KUKA KRL program: EPS_2_251692_SAMH01_A_20251205090654.src

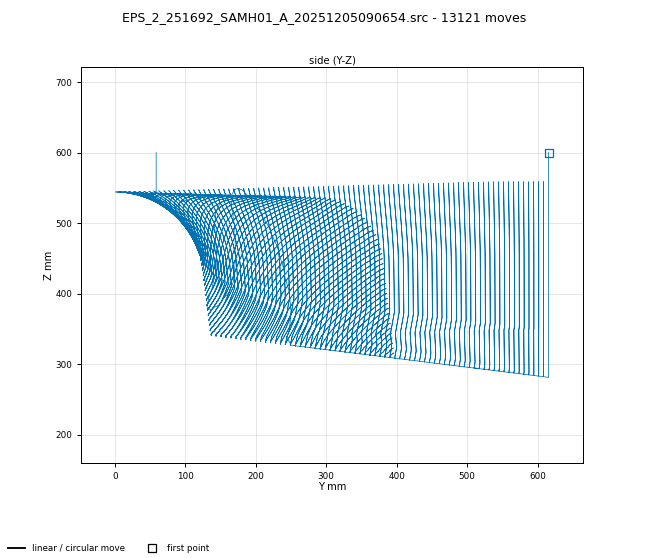
[picture p0: tool path of EPS_2_251692_SAMH01_A_20251205090654.src, 13121 of 13123 moves have a stored position in this frame; points joined in program order, loops and branches not executed]
&ACCESS RVP
&REL 4
&COMMENT QRS 19112012
&PARAM EDITMASK = *
DEF PART()
EXT BAS (BAS_COMMAND :IN,REAL :IN )
INT I
BAS (#INITMOV,0 )

;KUKA QRS Post kuka4.cps  Date:22-06-2017 !

File_ID=2943

QRS_PRE_INIT()

;Init var - Until changes are made in qrs_pre_init
Outlet_Square_prg=0
Inlet_1_Square_prg=0
Inlet_2_Square_prg=0
Inlet_3_Square_prg=0
Inlet_4_Square_prg=0
Inlet_5_Square_prg=0

Outlet_1={X 0.000, Y 535.490, Z 458.500, B 0.000, E1 0.000 }
Inlet_1={X 0.000, Y 556.400, Z 433.500, B 0.000, E1 180.000 }
Outlet_1_type=201
Inlet_1_type=0
;QRS#1=Sidecore dimensions
;QRS#2=200-8" PVC SDR 35
;QRS#3=DeadEnd 201
;QRS#4=
;QRS#5=
;QRS#6=
;QRS#7=
;QRS#8=
;QRS#9=12-08 PSX
;QRS#10=

;QRS#11=
;QRS#12=
;QRS#13=
;QRS#14=
;QRS#15=
;QRS#16=1220x127x838 2,75'
;QRS#17=EPS Height
;QRS#18=559
;QRS#19=*
;QRS#20= UPDATED VERSION 22-06-2017
;QRS#21=*
Outlet_Square=0100
Inlet_1_Square=00
Inlet_2_Square=0
Inlet_3_Square=0
Inlet_4_Square=0
Inlet_5_Square=0
Mill_Square=1
Outlet_Square_Prg=204
Inlet_1_Square_prg=0

QRS_INIT()

$ADVANCE=5

; T1
PTP {E1 173.595,E2 173.595}
PTP {X 0,Y 615.506,A -85,B 0,C 180,E1 173.595,E2 173.595,E3 0,E4 0,E5 0,E6 0}
QRS_SPEED_INIT()
LIN {X 0,Y 615.506,Z 600,A -85,B 0,C 180,E1 173.595,E2 173.595,E3 0,E4 0,E5 0,E6 0} C_VEL
LIN {X 0,Y 615.506,Z 291.363,A -85,B 0,C 180,E1 173.595,E2 173.595} C_VEL
LIN {X 0,Y 615.506,Z 283.186,A -85,B 0,C 180,E1 173.595,E2 173.595} C_VEL
LIN {X 0,Y 615.49,Z 281.186,A -85,B 0,C 180,E1 173.408,E2 173.408} C_VEL
LIN {X 0,Y 615.486,Z 281.199,A -85,B 0,C 180,E1 170.802,E2 170.802} C_VEL
LIN {X 0,Y 615.467,Z 281.188,A -85,B 0,C 180,E1 168.139,E2 168.139} C_VEL
LIN {X 0,Y 615.487,Z 281.188,A -85,B 0,C 180,E1 165.451,E2 165.451} C_VEL
LIN {X 0,Y 615.474,Z 281.196,A -85,B 0,C 180,E1 162.73,E2 162.73} C_VEL
LIN {X 0,Y 615.487,Z 281.182,A -85,B 0,C 180,E1 159.968,E2 159.968} C_VEL
LIN {X 0,Y 615.487,Z 281.2,A -85,B 0,C 180,E1 157.156,E2 157.156} C_VEL
LIN {X 0,Y 615.469,Z 281.189,A -85,B 0,C 180,E1 154.432,E2 154.432} C_VEL
LIN {X 0,Y 615.482,Z 281.184,A -85,B 0,C 180,E1 152.085,E2 152.085} C_VEL
LIN {X 0,Y 615.489,Z 281.198,A -85,B 0,C 180,E1 149.081,E2 149.081} C_VEL
LIN {X 0,Y 615.472,Z 281.187,A -85,B 0,C 180,E1 146.466,E2 146.466} C_VEL
LIN {X 0,Y 615.492,Z 281.181,A -85,B 0,C 180,E1 144.164,E2 144.164} C_VEL
LIN {X 0,Y 615.485,Z 281.186,A -85,B 0,C 180,E1 141.932,E2 141.932} C_VEL
LIN {X 0,Y 615.485,Z 281.201,A -85,B 0,C 180,E1 139.394,E2 139.394} C_VEL
LIN {X 0,Y 615.471,Z 281.189,A -85,B 0,C 180,E1 136.754,E2 136.754} C_VEL
LIN {X 0,Y 615.486,Z 281.186,A -85,B 0,C 180,E1 133.998,E2 133.998} C_VEL
LIN {X 0,Y 615.497,Z 281.199,A -85,B 0,C 180,E1 131.472,E2 131.472} C_VEL
LIN {X 0,Y 615.472,Z 281.19,A -85,B 0,C 180,E1 128.904,E2 128.904} C_VEL
LIN {X 0,Y 615.484,Z 281.183,A -85,B 0,C 180,E1 126.424,E2 126.424} C_VEL
LIN {X 0,Y 615.495,Z 281.201,A -85,B 0,C 180,E1 123.536,E2 123.536} C_VEL
LIN {X 0,Y 615.474,Z 281.188,A -85,B 0,C 180,E1 120.92,E2 120.92} C_VEL
LIN {X 0,Y 615.491,Z 281.182,A -85,B 0,C 180,E1 118.452,E2 118.452} C_VEL
LIN {X 0,Y 615.492,Z 281.199,A -85,B 0,C 180,E1 115.571,E2 115.571} C_VEL
LIN {X 0,Y 615.48,Z 281.184,A -85,B 0,C 180,E1 112.844,E2 112.844} C_VEL
LIN {X 0,Y 615.483,Z 281.193,A -85,B 0,C 180,E1 110.032,E2 110.032} C_VEL
LIN {X 0,Y 615.475,Z 281.19,A -85,B 0,C 180,E1 107.27,E2 107.27} C_VEL
LIN {X 0,Y 615.482,Z 281.185,A -85,B 0,C 180,E1 104.549,E2 104.549} C_VEL
LIN {X 0,Y 615.486,Z 281.202,A -85,B 0,C 180,E1 101.861,E2 101.861} C_VEL
LIN {X 0,Y 615.479,Z 281.187,A -85,B 0,C 180,E1 99.199,E2 99.199} C_VEL
LIN {X 0,Y 615.479,Z 281.187,A -85,B 0,C 180,E1 96.557,E2 96.557} C_VEL
LIN {X 0,Y 615.486,Z 281.203,A -85,B 0,C 180,E1 93.928,E2 93.928} C_VEL
LIN {X 0,Y 615.48,Z 281.186,A -85,B 0,C 180,E1 91.309,E2 91.309} C_VEL
LIN {X 0,Y 615.48,Z 281.186,A -85,B 0,C 180,E1 88.691,E2 88.691} C_VEL
LIN {X 0,Y 615.486,Z 281.203,A -85,B 0,C 180,E1 86.072,E2 86.072} C_VEL
LIN {X 0,Y 615.48,Z 281.186,A -85,B 0,C 180,E1 83.424,E2 83.424} C_VEL
LIN {X 0,Y 615.479,Z 281.187,A -85,B 0,C 180,E1 80.801,E2 80.801} C_VEL
LIN {X 0,Y 615.486,Z 281.202,A -85,B 0,C 180,E1 78.139,E2 78.139} C_VEL
LIN {X 0,Y 615.482,Z 281.185,A -85,B 0,C 180,E1 75.451,E2 75.451} C_VEL
LIN {X 0,Y 615.475,Z 281.19,A -85,B 0,C 180,E1 72.73,E2 72.73} C_VEL
LIN {X 0,Y 615.483,Z 281.193,A -85,B 0,C 180,E1 69.968,E2 69.968} C_VEL
LIN {X 0,Y 615.481,Z 281.184,A -85,B 0,C 180,E1 67.156,E2 67.156} C_VEL
LIN {X 0,Y 615.495,Z 281.199,A -85,B 0,C 180,E1 64.285,E2 64.285} C_VEL
LIN {X 0,Y 615.483,Z 281.183,A -85,B 0,C 180,E1 61.342,E2 61.342} C_VEL
LIN {X 0,Y 615.473,Z 281.191,A -85,B 0,C 180,E1 58.915,E2 58.915} C_VEL
LIN {X 0,Y 615.495,Z 281.201,A -85,B 0,C 180,E1 56.464,E2 56.464} C_VEL
LIN {X 0,Y 615.484,Z 281.183,A -85,B 0,C 180,E1 53.576,E2 53.576} C_VEL
LIN {X 0,Y 615.474,Z 281.193,A -85,B 0,C 180,E1 50.939,E2 50.939} C_VEL
LIN {X 0,Y 615.497,Z 281.199,A -85,B 0,C 180,E1 48.528,E2 48.528} C_VEL
LIN {X 0,Y 615.492,Z 281.183,A -85,B 0,C 180,E1 45.852,E2 45.852} C_VEL
LIN {X 0,Y 615.473,Z 281.193,A -85,B 0,C 180,E1 43.047,E2 43.047} C_VEL
LIN {X 0,Y 615.485,Z 281.201,A -85,B 0,C 180,E1 40.606,E2 40.606} C_VEL
LIN {X 0,Y 615.485,Z 281.185,A -85,B 0,C 180,E1 38.013,E2 38.013} C_VEL
LIN {X 0,Y 615.476,Z 281.185,A -85,B 0,C 180,E1 35.616,E2 35.616} C_VEL
LIN {X 0,Y 615.47,Z 281.192,A -85,B 0,C 180,E1 33.237,E2 33.237} C_VEL
LIN {X 0,Y 615.489,Z 281.198,A -85,B 0,C 180,E1 30.919,E2 30.919} C_VEL
LIN {X 0,Y 615.484,Z 281.183,A -85,B 0,C 180,E1 27.915,E2 27.915} C_VEL
LIN {X 0,Y 615.467,Z 281.189,A -85,B 0,C 180,E1 25.568,E2 25.568} C_VEL
LIN {X 0,Y 615.487,Z 281.2,A -85,B 0,C 180,E1 22.844,E2 22.844} C_VEL
LIN {X 0,Y 615.487,Z 281.182,A -85,B 0,C 180,E1 20.032,E2 20.032} C_VEL
LIN {X 0,Y 615.474,Z 281.196,A -85,B 0,C 180,E1 17.27,E2 17.27} C_VEL
LIN {X 0,Y 615.487,Z 281.188,A -85,B 0,C 180,E1 14.549,E2 14.549} C_VEL
LIN {X 0,Y 615.467,Z 281.188,A -85,B 0,C 180,E1 11.861,E2 11.861} C_VEL
LIN {X 0,Y 615.486,Z 281.199,A -85,B 0,C 180,E1 9.198,E2 9.198} C_VEL
LIN {X 0,Y 615.491,Z 281.185,A -85,B 0,C 180,E1 6.556,E2 6.556} C_VEL
LIN {X 0,Y 615.464,Z 281.189,A -85,B 0,C 180,E1 3.928,E2 3.928} C_VEL
LIN {X 0,Y 615.485,Z 281.2,A -85,B 0,C 180,E1 1.308,E2 1.308} C_VEL
LIN {X 0,Y 615.491,Z 281.186,A -85,B 0,C 180,E1 -1.309,E2 -1.309} C_VEL
LIN {X 0,Y 615.465,Z 281.188,A -85,B 0,C 180,E1 -3.929,E2 -3.929} C_VEL
LIN {X 0,Y 615.483,Z 281.2,A -85,B 0,C 180,E1 -6.586,E2 -6.586} C_VEL
LIN {X 0,Y 615.492,Z 281.185,A -85,B 0,C 180,E1 -9.199,E2 -9.199} C_VEL
LIN {X 0,Y 615.462,Z 281.19,A -85,B 0,C 180,E1 -11.862,E2 -11.862} C_VEL
LIN {X 0,Y 615.487,Z 281.202,A -85,B 0,C 180,E1 -14.549,E2 -14.549} C_VEL
LIN {X 0,Y 615.491,Z 281.183,A -85,B 0,C 180,E1 -17.271,E2 -17.271} C_VEL
LIN {X 0,Y 615.463,Z 281.194,A -85,B 0,C 180,E1 -20.034,E2 -20.034} C_VEL
LIN {X 0,Y 615.491,Z 281.19,A -85,B 0,C 180,E1 -22.845,E2 -22.845} C_VEL
LIN {X 0,Y 615.458,Z 281.189,A -85,B 0,C 180,E1 -25.566,E2 -25.566} C_VEL
LIN {X 0,Y 615.462,Z 281.194,A -85,B 0,C 180,E1 -27.917,E2 -27.917} C_VEL
LIN {X 0,Y 615.474,Z 281.199,A -85,B 0,C 180,E1 -30.161,E2 -30.161} C_VEL
LIN {X 0,Y 615.494,Z 281.197,A -85,B 0,C 180,E1 -32.457,E2 -32.457} C_VEL
LIN {X 0,Y 615.494,Z 281.186,A -85,B 0,C 180,E1 -34.815,E2 -34.815} C_VEL
LIN {X 0,Y 615.466,Z 281.187,A -85,B 0,C 180,E1 -37.244,E2 -37.244} C_VEL
LIN {X 0,Y 615.485,Z 281.198,A -85,B 0,C 180,E1 -40.09,E2 -40.09} C_VEL
LIN {X 0,Y 615.472,Z 281.186,A -85,B 0,C 180,E1 -43.047,E2 -43.047} C_VEL
LIN {X 0,Y 615.469,Z 281.197,A -85,B 0,C 180,E1 -45.85,E2 -45.85} C_VEL
LIN {X 0,Y 615.493,Z 281.188,A -85,B 0,C 180,E1 -48.528,E2 -48.528} C_VEL
LIN {X 0,Y 615.46,Z 281.188,A -85,B 0,C 180,E1 -51.095,E2 -51.095} C_VEL
LIN {X 0,Y 615.459,Z 281.195,A -85,B 0,C 180,E1 -53.574,E2 -53.574} C_VEL
LIN {X 0,Y 615.496,Z 281.187,A -85,B 0,C 180,E1 -56.465,E2 -56.465} C_VEL
LIN {X 0,Y 615.455,Z 281.19,A -85,B 0,C 180,E1 -59.079,E2 -59.079} C_VEL
LIN {X 0,Y 615.463,Z 281.196,A -85,B 0,C 180,E1 -61.554,E2 -61.554} C_VEL
LIN {X 0,Y 615.498,Z 281.185,A -85,B 0,C 180,E1 -64.43,E2 -64.43} C_VEL
LIN {X 0,Y 615.497,Z 281.361,A -85,B 0,C 180,E1 -65.958,E2 -65.958} C_VEL
LIN {X 0,Y 615.494,Z 296.441,A -85,B 0,C 180,E1 -68.569,E2 -68.569} C_VEL
LIN {X 0,Y 615.488,Z 313.211,A -85,B 0,C 180,E1 -71.396,E2 -71.396} C_VEL
LIN {X 0,Y 615.498,Z 330.499,A -85,B 0,C 180,E1 -74.265,E2 -74.265} C_VEL
LIN {X 0,Y 615.496,Z 347.73,A -85,B 0,C 180,E1 -77.072,E2 -77.072} C_VEL
LIN {X 0,Y 615.493,Z 349.262,A -85,B 0,C 180,E1 -77.156,E2 -77.156} C_VEL
LIN {X 0,Y 615.497,Z 454.843,A -85,B 0,C 180,E1 -78.411,E2 -78.411} C_VEL
LIN {X 0,Y 615.499,Z 467.352,A -85,B 0,C 180,E1 -78.682,E2 -78.682} C_VEL
LIN {X 0,Y 615.496,Z 480.501,A -85,B 0,C 180,E1 -79.109,E2 -79.109} C_VEL
LIN {X 0,Y 615.486,Z 492.482,A -85,B 0,C 180,E1 -79.64,E2 -79.64} C_VEL
LIN {X 0,Y 615.493,Z 503.998,A -85,B 0,C 180,E1 -80.304,E2 -80.304} C_VEL
LIN {X 0,Y 615.499,Z 514.344,A -85,B 0,C 180,E1 -81.05,E2 -81.05} C_VEL
LIN {X 0,Y 615.497,Z 522.814,A -85,B 0,C 180,E1 -81.794,E2 -81.794} C_VEL
LIN {X 0,Y 615.498,Z 530.608,A -85,B 0,C 180,E1 -82.62,E2 -82.62} C_VEL
LIN {X 0,Y 615.496,Z 538.204,A -85,B 0,C 180,E1 -83.608,E2 -83.608} C_VEL
LIN {X 0,Y 615.498,Z 545.205,A -85,B 0,C 180,E1 -84.759,E2 -84.759} C_VEL
LIN {X 0,Y 615.493,Z 549.852,A -85,B 0,C 180,E1 -85.744,E2 -85.744} C_VEL
LIN {X 0,Y 615.495,Z 553.399,A -85,B 0,C 180,E1 -86.727,E2 -86.727} C_VEL
LIN {X 0,Y 615.497,Z 555.233,A -85,B 0,C 180,E1 -87.382,E2 -87.382} C_VEL
LIN {X 0,Y 615.499,Z 556.608,A -85,B 0,C 180,E1 -88.037,E2 -88.037} C_VEL
LIN {X 0,Y 615.496,Z 558.174,A -85,B 0,C 180,E1 -89.346,E2 -89.346} C_VEL
LIN {X 0,Y 615.494,Z 558.389,A -85,B 0,C 180,E1 -90,E2 -90} C_VEL
LIN {X 0,Y 615.496,Z 557.58,A -85,B 0,C 180,E1 -91.309,E2 -91.309} C_VEL
LIN {X 0,Y 615.499,Z 556.608,A -85,B 0,C 180,E1 -91.963,E2 -91.963} C_VEL
LIN {X 0,Y 615.497,Z 555.233,A -85,B 0,C 180,E1 -92.618,E2 -92.618} C_VEL
LIN {X 0,Y 615.496,Z 552.35,A -85,B 0,C 180,E1 -93.601,E2 -93.601} C_VEL
LIN {X 0,Y 615.498,Z 548.442,A -85,B 0,C 180,E1 -94.584,E2 -94.584} C_VEL
LIN {X 0,Y 615.499,Z 543.406,A -85,B 0,C 180,E1 -95.57,E2 -95.57} C_VEL
LIN {X 0,Y 615.497,Z 536.87,A -85,B 0,C 180,E1 -96.583,E2 -96.583} C_VEL
LIN {X 0,Y 615.497,Z 529.135,A -85,B 0,C 180,E1 -97.545,E2 -97.545} C_VEL
LIN {X 0,Y 615.498,Z 521.047,A -85,B 0,C 180,E1 -98.371,E2 -98.371} C_VEL
LIN {X 0,Y 615.499,Z 511.17,A -85,B 0,C 180,E1 -99.198,E2 -99.198} C_VEL
LIN {X 0,Y 615.493,Z 499.985,A -85,B 0,C 180,E1 -99.945,E2 -99.945} C_VEL
LIN {X 0,Y 615.489,Z 489.027,A -85,B 0,C 180,E1 -100.527,E2 -100.527} C_VEL
LIN {X 0,Y 615.499,Z 476.422,A -85,B 0,C 180,E1 -101.042,E2 -101.042} C_VEL
LIN {X 0,Y 615.499,Z 464.075,A -85,B 0,C 180,E1 -101.401,E2 -101.401} C_VEL
LIN {X 0,Y 615.498,Z 450.483,A -85,B 0,C 180,E1 -101.651,E2 -101.651} C_VEL
LIN {X 0,Y 615.494,Z 348.55,A -85,B 0,C 180,E1 -102.865,E2 -102.865} C_VEL
LIN {X 0,Y 615.495,Z 346.987,A -85,B 0,C 180,E1 -103.033,E2 -103.033} C_VEL
LIN {X 0,Y 615.495,Z 329.466,A -85,B 0,C 180,E1 -105.905,E2 -105.905} C_VEL
LIN {X 0,Y 615.487,Z 312.962,A -85,B 0,C 180,E1 -108.646,E2 -108.646} C_VEL
LIN {X 0,Y 615.494,Z 296.441,A -85,B 0,C 180,E1 -111.431,E2 -111.431} C_VEL
LIN {X 0,Y 615.497,Z 281.361,A -85,B 0,C 180,E1 -114.042,E2 -114.042} C_VEL
LIN {X 0,Y 615.465,Z 281.196,A -85,B 0,C 180,E1 -116.444,E2 -116.444} C_VEL
LIN {X 0,Y 615.453,Z 281.193,A -85,B 0,C 180,E1 -118.659,E2 -118.659} C_VEL
LIN {X 0,Y 615.462,Z 281.188,A -85,B 0,C 180,E1 -121.082,E2 -121.082} C_VEL
LIN {X 0,Y 615.491,Z 281.201,A -85,B 0,C 180,E1 -124.021,E2 -124.021} C_VEL
LIN {X 0,Y 615.459,Z 281.195,A -85,B 0,C 180,E1 -126.426,E2 -126.426} C_VEL
LIN {X 0,Y 615.47,Z 281.187,A -85,B 0,C 180,E1 -129.06,E2 -129.06} C_VEL
LIN {X 0,Y 615.478,Z 281.198,A -85,B 0,C 180,E1 -132.079,E2 -132.079} C_VEL
LIN {X 0,Y 615.47,Z 281.196,A -85,B 0,C 180,E1 -134.15,E2 -134.15} C_VEL
LIN {X 0,Y 615.472,Z 281.186,A -85,B 0,C 180,E1 -136.953,E2 -136.953} C_VEL
LIN {X 0,Y 615.485,Z 281.198,A -85,B 0,C 180,E1 -139.91,E2 -139.91} C_VEL
LIN {X 0,Y 615.466,Z 281.187,A -85,B 0,C 180,E1 -142.756,E2 -142.756} C_VEL
LIN {X 0,Y 615.492,Z 281.189,A -85,B 0,C 180,E1 -145.297,E2 -145.297} C_VEL
LIN {X 0,Y 615.494,Z 281.201,A -85,B 0,C 180,E1 -147.666,E2 -147.666} C_VEL
LIN {X 0,Y 615.459,Z 281.193,A -85,B 0,C 180,E1 -150.208,E2 -150.208} C_VEL
LIN {X 0,Y 615.497,Z 281.183,A -85,B 0,C 180,E1 -152.951,E2 -152.951} C_VEL
LIN {X 0,Y 615.482,Z 281.198,A -85,B 0,C 180,E1 -155.727,E2 -155.727} C_VEL
LIN {X 0,Y 615.469,Z 281.196,A -85,B 0,C 180,E1 -157.863,E2 -157.863} C_VEL
LIN {X 0,Y 615.483,Z 281.184,A -85,B 0,C 180,E1 -160.662,E2 -160.662} C_VEL
LIN {X 0,Y 615.482,Z 281.2,A -85,B 0,C 180,E1 -163.566,E2 -163.566} C_VEL
LIN {X 0,Y 615.461,Z 281.19,A -85,B 0,C 180,E1 -166.125,E2 -166.125} C_VEL
LIN {X 0,Y 615.493,Z 281.185,A -85,B 0,C 180,E1 -168.807,E2 -168.807} C_VEL
LIN {X 0,Y 615.487,Z 281.198,A -85,B 0,C 180,E1 -171.463,E2 -171.463} C_VEL
LIN {X 0,Y 615.464,Z 281.188,A -85,B 0,C 180,E1 -174.101,E2 -174.101} C_VEL
LIN {X 0,Y 615.489,Z 281.186,A -85,B 0,C 180,E1 -176.727,E2 -176.727} C_VEL
LIN {X 0,Y 615.489,Z 281.198,A -85,B 0,C 180,E1 -179.345,E2 -179.345} C_VEL
LIN {X 0,Y 615.465,Z 281.189,A -85,B 0,C 180,E1 -181.963,E2 -181.963} C_VEL
LIN {X 0,Y 615.492,Z 281.185,A -85,B 0,C 180,E1 -184.584,E2 -184.584} C_VEL
LIN {X 0,Y 615.49,Z 281.186,A -85,B 0,C 180,E1 -186.592,E2 -186.592} C_VEL
LIN {X 0,Y 614.813,Z 281.345,A -85,B 0,C 180,E1 -187.138,E2 -187.138} C_VEL
LIN {X 0,Y 611.978,Z 281.748,A -85,B 0,C 180,E1 -188.024,E2 -188.024} C_VEL
LIN {X 0,Y 609.584,Z 282.063,A -85,B 0,C 180,E1 -188.736,E2 -188.736} C_VEL
LIN {X 0,Y 608.544,Z 282.183,A -85,B 0,C 180,E1 -189.286,E2 -189.286} C_VEL
LIN {X 0,Y 608.452,Z 282.191,A -85,B 0,C 180,E1 -189.472,E2 -189.472} C_VEL
LIN {X 0,Y 608.448,Z 282.188,A -85,B 0,C 180,E1 -192,E2 -192} C_VEL
LIN {X 0,Y 608.473,Z 282.19,A -85,B 0,C 180,E1 -194.72,E2 -194.72} C_VEL
LIN {X 0,Y 608.441,Z 282.191,A -85,B 0,C 180,E1 -197.476,E2 -197.476} C_VEL
LIN {X 0,Y 608.462,Z 282.187,A -85,B 0,C 180,E1 -200.274,E2 -200.274} C_VEL
LIN {X 0,Y 608.443,Z 282.195,A -85,B 0,C 180,E1 -203.124,E2 -203.124} C_VEL
LIN {X 0,Y 608.457,Z 282.187,A -85,B 0,C 180,E1 -205.721,E2 -205.721} C_VEL
LIN {X 0,Y 608.448,Z 282.19,A -85,B 0,C 180,E1 -208.266,E2 -208.266} C_VEL
LIN {X 0,Y 608.473,Z 282.191,A -85,B 0,C 180,E1 -210.544,E2 -210.544} C_VEL
LIN {X 0,Y 608.447,Z 282.197,A -85,B 0,C 180,E1 -212.88,E2 -212.88} C_VEL
LIN {X 0,Y 608.44,Z 282.191,A -85,B 0,C 180,E1 -215.277,E2 -215.277} C_VEL
LIN {X 0,Y 608.464,Z 282.189,A -85,B 0,C 180,E1 -218.242,E2 -218.242} C_VEL
LIN {X 0,Y 608.472,Z 282.19,A -85,B 0,C 180,E1 -220.333,E2 -220.333} C_VEL
LIN {X 0,Y 608.46,Z 282.188,A -85,B 0,C 180,E1 -223.309,E2 -223.309} C_VEL
LIN {X 0,Y 608.469,Z 282.188,A -85,B 0,C 180,E1 -226.132,E2 -226.132} C_VEL
LIN {X 0,Y 608.449,Z 282.194,A -85,B 0,C 180,E1 -228.824,E2 -228.824} C_VEL
LIN {X 0,Y 608.46,Z 282.187,A -85,B 0,C 180,E1 -231.412,E2 -231.412} C_VEL
LIN {X 0,Y 608.472,Z 282.187,A -85,B 0,C 180,E1 -233.951,E2 -233.951} C_VEL
LIN {X 0,Y 608.467,Z 282.194,A -85,B 0,C 180,E1 -236.33,E2 -236.33} C_VEL
LIN {X 0,Y 608.47,Z 282.191,A -85,B 0,C 180,E1 -238.728,E2 -238.728} C_VEL
LIN {X 0,Y 608.471,Z 282.185,A -85,B 0,C 180,E1 -241.379,E2 -241.379} C_VEL
LIN {X 0,Y 608.476,Z 282.194,A -85,B 0,C 180,E1 -244.277,E2 -244.277} C_VEL
LIN {X 0,Y 608.447,Z 282.19,A -85,B 0,C 180,E1 -246.876,E2 -246.876} C_VEL
LIN {X 0,Y 608.461,Z 282.189,A -85,B 0,C 180,E1 -249.726,E2 -249.726} C_VEL
LIN {X 0,Y 608.446,Z 282.194,A -85,B 0,C 180,E1 -252.524,E2 -252.524} C_VEL
LIN {X 0,Y 608.47,Z 282.185,A -85,B 0,C 180,E1 -255.28,E2 -255.28} C_VEL
LIN {X 0,Y 608.461,Z 282.194,A -85,B 0,C 180,E1 -258.001,E2 -258.001} C_VEL
LIN {X 0,Y 608.466,Z 282.188,A -85,B 0,C 180,E1 -260.694,E2 -260.694} C_VEL
LIN {X 0,Y 608.475,Z 282.186,A -85,B 0,C 180,E1 -263.368,E2 -263.368} C_VEL
LIN {X 0,Y 608.454,Z 282.198,A -85,B 0,C 180,E1 -266.026,E2 -266.026} C_VEL
LIN {X 0,Y 608.465,Z 282.187,A -85,B 0,C 180,E1 -268.676,E2 -268.676} C_VEL
LIN {X 0,Y 608.465,Z 282.187,A -85,B 0,C 180,E1 -271.324,E2 -271.324} C_VEL
LIN {X 0,Y 608.454,Z 282.198,A -85,B 0,C 180,E1 -273.974,E2 -273.974} C_VEL
LIN {X 0,Y 608.475,Z 282.186,A -85,B 0,C 180,E1 -276.632,E2 -276.632} C_VEL
LIN {X 0,Y 608.466,Z 282.188,A -85,B 0,C 180,E1 -279.306,E2 -279.306} C_VEL
LIN {X 0,Y 608.461,Z 282.194,A -85,B 0,C 180,E1 -281.999,E2 -281.999} C_VEL
LIN {X 0,Y 608.47,Z 282.185,A -85,B 0,C 180,E1 -284.72,E2 -284.72} C_VEL
LIN {X 0,Y 608.446,Z 282.194,A -85,B 0,C 180,E1 -287.476,E2 -287.476} C_VEL
LIN {X 0,Y 608.461,Z 282.189,A -85,B 0,C 180,E1 -290.274,E2 -290.274} C_VEL
LIN {X 0,Y 608.446,Z 282.19,A -85,B 0,C 180,E1 -293.124,E2 -293.124} C_VEL
LIN {X 0,Y 608.476,Z 282.194,A -85,B 0,C 180,E1 -295.723,E2 -295.723} C_VEL
LIN {X 0,Y 608.473,Z 282.185,A -85,B 0,C 180,E1 -298.621,E2 -298.621} C_VEL
LIN {X 0,Y 608.47,Z 282.191,A -85,B 0,C 180,E1 -301.315,E2 -301.315} C_VEL
LIN {X 0,Y 608.475,Z 282.191,A -85,B 0,C 180,E1 -303.736,E2 -303.736} C_VEL
LIN {X 0,Y 608.471,Z 282.187,A -85,B 0,C 180,E1 -306.09,E2 -306.09} C_VEL
LIN {X 0,Y 608.46,Z 282.187,A -85,B 0,C 180,E1 -308.588,E2 -308.588} C_VEL
LIN {X 0,Y 608.463,Z 282.195,A -85,B 0,C 180,E1 -311.343,E2 -311.343} C_VEL
LIN {X 0,Y 608.458,Z 282.187,A -85,B 0,C 180,E1 -314.265,E2 -314.265} C_VEL
LIN {X 0,Y 608.441,Z 282.194,A -85,B 0,C 180,E1 -317.04,E2 -317.04} C_VEL
LIN {X 0,Y 608.451,Z 282.192,A -85,B 0,C 180,E1 -319.697,E2 -319.697} C_VEL
LIN {X 0,Y 608.463,Z 282.186,A -85,B 0,C 180,E1 -322.254,E2 -322.254} C_VEL
LIN {X 0,Y 608.481,Z 282.191,A -85,B 0,C 180,E1 -325.088,E2 -325.088} C_VEL
LIN {X 0,Y 608.46,Z 282.187,A -85,B 0,C 180,E1 -327.906,E2 -327.906} C_VEL
LIN {X 0,Y 608.466,Z 282.186,A -85,B 0,C 180,E1 -330.221,E2 -330.221} C_VEL
LIN {X 0,Y 608.469,Z 282.19,A -85,B 0,C 180,E1 -332.792,E2 -332.792} C_VEL
LIN {X 0,Y 608.481,Z 282.184,A -85,B 0,C 180,E1 -335.844,E2 -335.844} C_VEL
LIN {X 0,Y 608.46,Z 282.187,A -85,B 0,C 180,E1 -338.309,E2 -338.309} C_VEL
LIN {X 0,Y 608.448,Z 282.197,A -85,B 0,C 180,E1 -341.131,E2 -341.131} C_VEL
LIN {X 0,Y 608.454,Z 282.187,A -85,B 0,C 180,E1 -343.906,E2 -343.906} C_VEL
LIN {X 0,Y 608.457,Z 282.192,A -85,B 0,C 180,E1 -346.644,E2 -346.644} C_VEL
LIN {X 0,Y 608.468,Z 282.188,A -85,B 0,C 180,E1 -349.351,E2 -349.351} C_VEL
LIN {X 0,Y 608.46,Z 282.186,A -85,B 0,C 180,E1 -352.033,E2 -352.033} C_VEL
LIN {X 0,Y 608.463,Z 282.194,A -85,B 0,C 180,E1 -354.699,E2 -354.699} C_VEL
LIN {X 0,Y 608.481,Z 282.186,A -85,B 0,C 180,E1 -357.352,E2 -357.352} C_VEL
LIN {X 0,Y 608.457,Z 282.187,A -85,B 0,C 180,E1 -360,E2 -360} C_VEL
LIN {X 0,Y 608.474,Z 282.194,A -85,B 0,C 180,E1 -362.648,E2 -362.648} C_VEL
LIN {X 0,Y 608.467,Z 282.187,A -85,B 0,C 180,E1 -365.302,E2 -365.302} C_VEL
LIN {X 0,Y 608.46,Z 282.187,A -85,B 0,C 180,E1 -367.968,E2 -367.968} C_VEL
LIN {X 0,Y 608.463,Z 282.196,A -85,B 0,C 180,E1 -370.65,E2 -370.65} C_VEL
LIN {X 0,Y 608.464,Z 282.186,A -85,B 0,C 180,E1 -373.357,E2 -373.357} C_VEL
LIN {X 0,Y 608.442,Z 282.192,A -85,B 0,C 180,E1 -376.095,E2 -376.095} C_VEL
LIN {X 0,Y 608.455,Z 282.191,A -85,B 0,C 180,E1 -378.87,E2 -378.87} C_VEL
LIN {X 0,Y 608.452,Z 282.188,A -85,B 0,C 180,E1 -381.693,E2 -381.693} C_VEL
LIN {X 0,Y 608.453,Z 282.195,A -85,B 0,C 180,E1 -384.571,E2 -384.571} C_VEL
LIN {X 0,Y 608.439,Z 282.189,A -85,B 0,C 180,E1 -387.519,E2 -387.519} C_VEL
LIN {X 0,Y 608.447,Z 282.192,A -85,B 0,C 180,E1 -389.97,E2 -389.97} C_VEL
LIN {X 0,Y 608.453,Z 282.189,A -85,B 0,C 180,E1 -392.88,E2 -392.88} C_VEL
LIN {X 0,Y 608.429,Z 282.19,A -85,B 0,C 180,E1 -395.279,E2 -395.279} C_VEL
LIN {X 0,Y 608.457,Z 282.189,A -85,B 0,C 180,E1 -397.748,E2 -397.748} C_VEL
LIN {X 0,Y 608.451,Z 282.196,A -85,B 0,C 180,E1 -400.331,E2 -400.331} C_VEL
LIN {X 0,Y 608.442,Z 282.189,A -85,B 0,C 180,E1 -402.961,E2 -402.961} C_VEL
LIN {X 0,Y 608.44,Z 282.193,A -85,B 0,C 180,E1 -405.738,E2 -405.738} C_VEL
LIN {X 0,Y 608.457,Z 282.194,A -85,B 0,C 180,E1 -407.94,E2 -407.94} C_VEL
LIN {X 0,Y 608.44,Z 282.19,A -85,B 0,C 180,E1 -410.706,E2 -410.706} C_VEL
LIN {X 0,Y 608.431,Z 282.19,A -85,B 0,C 180,E1 -413.084,E2 -413.084} C_VEL
LIN {X 0,Y 608.45,Z 282.19,A -85,B 0,C 180,E1 -415.53,E2 -415.53} C_VEL
LIN {X 0,Y 608.458,Z 282.196,A -85,B 0,C 180,E1 -417.906,E2 -417.906} C_VEL
LIN {X 0,Y 608.477,Z 282.19,A -85,B 0,C 180,E1 -420.222,E2 -420.222} C_VEL
LIN {X 0,Y 608.423,Z 282.192,A -85,B 0,C 180,E1 -423.225,E2 -423.225} C_VEL
LIN {X 0,Y 608.496,Z 282.338,A -85,B 0,C 180,E1 -425.844,E2 -425.844} C_VEL
LIN {X 0,Y 608.54,Z 296.465,A -85,B 0,C 180,E1 -428.312,E2 -428.312} C_VEL
LIN {X 0,Y 608.514,Z 313.852,A -85,B 0,C 180,E1 -431.273,E2 -431.273} C_VEL
LIN {X 0,Y 608.501,Z 330.613,A -85,B 0,C 180,E1 -434.08,E2 -434.08} C_VEL
LIN {X 0,Y 608.495,Z 348.253,A -85,B 0,C 180,E1 -436.963,E2 -436.963} C_VEL
LIN {X 0,Y 608.589,Z 350.746,A -85,B 0,C 180,E1 -437.029,E2 -437.029} C_VEL
LIN {X 0,Y 608.548,Z 454.957,A -85,B 0,C 180,E1 -438.277,E2 -438.277} C_VEL
LIN {X 0,Y 608.547,Z 468.234,A -85,B 0,C 180,E1 -438.572,E2 -438.572} C_VEL
LIN {X 0,Y 608.54,Z 481.391,A -85,B 0,C 180,E1 -439.011,E2 -439.011} C_VEL
LIN {X 0,Y 608.507,Z 492.628,A -85,B 0,C 180,E1 -439.519,E2 -439.519} C_VEL
LIN {X 0,Y 608.487,Z 504.201,A -85,B 0,C 180,E1 -440.191,E2 -440.191} C_VEL
LIN {X 0,Y 608.485,Z 514.598,A -85,B 0,C 180,E1 -440.946,E2 -440.946} C_VEL
LIN {X 0,Y 608.475,Z 523.116,A -85,B 0,C 180,E1 -441.699,E2 -441.699} C_VEL
LIN {X 0,Y 608.471,Z 530.961,A -85,B 0,C 180,E1 -442.534,E2 -442.534} C_VEL
LIN {X 0,Y 608.461,Z 538.287,A -85,B 0,C 180,E1 -443.485,E2 -443.485} C_VEL
LIN {X 0,Y 608.45,Z 543.865,A -85,B 0,C 180,E1 -444.366,E2 -444.366} C_VEL
LIN {X 0,Y 608.432,Z 548.951,A -85,B 0,C 180,E1 -445.362,E2 -445.362} C_VEL
LIN {X 0,Y 608.449,Z 552.896,A -85,B 0,C 180,E1 -446.358,E2 -446.358} C_VEL
LIN {X 0,Y 608.425,Z 555.808,A -85,B 0,C 180,E1 -447.352,E2 -447.352} C_VEL
LIN {X 0,Y 608.444,Z 557.201,A -85,B 0,C 180,E1 -448.014,E2 -448.014} C_VEL
LIN {X 0,Y 608.438,Z 558.783,A -85,B 0,C 180,E1 -449.338,E2 -449.338} C_VEL
LIN {X 0,Y 608.434,Z 558.998,A -85,B 0,C 180,E1 -450,E2 -450} C_VEL
LIN {X 0,Y 608.448,Z 558.184,A -85,B 0,C 180,E1 -451.324,E2 -451.324} C_VEL
LIN {X 0,Y 608.444,Z 557.201,A -85,B 0,C 180,E1 -451.986,E2 -451.986} C_VEL
LIN {X 0,Y 608.425,Z 555.808,A -85,B 0,C 180,E1 -452.648,E2 -452.648} C_VEL
LIN {X 0,Y 608.449,Z 552.896,A -85,B 0,C 180,E1 -453.642,E2 -453.642} C_VEL
LIN {X 0,Y 608.432,Z 548.951,A -85,B 0,C 180,E1 -454.638,E2 -454.638} C_VEL
LIN {X 0,Y 608.45,Z 543.865,A -85,B 0,C 180,E1 -455.634,E2 -455.634} C_VEL
LIN {X 0,Y 608.442,Z 537.473,A -85,B 0,C 180,E1 -456.633,E2 -456.633} C_VEL
LIN {X 0,Y 608.475,Z 529.48,A -85,B 0,C 180,E1 -457.633,E2 -457.633} C_VEL
LIN {X 0,Y 608.487,Z 521.34,A -85,B 0,C 180,E1 -458.468,E2 -458.468} C_VEL
LIN {X 0,Y 608.485,Z 511.399,A -85,B 0,C 180,E1 -459.305,E2 -459.305} C_VEL
LIN {X 0,Y 608.506,Z 500.171,A -85,B 0,C 180,E1 -460.06,E2 -460.06} C_VEL
LIN {X 0,Y 608.516,Z 489.18,A -85,B 0,C 180,E1 -460.649,E2 -460.649} C_VEL
LIN {X 0,Y 608.535,Z 477.709,A -85,B 0,C 180,E1 -461.127,E2 -461.127} C_VEL
LIN {X 0,Y 608.55,Z 465.081,A -85,B 0,C 180,E1 -461.512,E2 -461.512} C_VEL
LIN {X 0,Y 608.564,Z 452.128,A -85,B 0,C 180,E1 -461.765,E2 -461.765} C_VEL
LIN {X 0,Y 608.531,Z 348.583,A -85,B 0,C 180,E1 -463.015,E2 -463.015} C_VEL
LIN {X 0,Y 608.491,Z 347.169,A -85,B 0,C 180,E1 -463.185,E2 -463.185} C_VEL
LIN {X 0,Y 608.491,Z 329.578,A -85,B 0,C 180,E1 -466.093,E2 -466.093} C_VEL
LIN {X 0,Y 608.507,Z 313.021,A -85,B 0,C 180,E1 -468.867,E2 -468.867} C_VEL
LIN {X 0,Y 608.542,Z 296.465,A -85,B 0,C 180,E1 -471.688,E2 -471.688} C_VEL
LIN {X 0,Y 608.503,Z 282.291,A -85,B 0,C 180,E1 -474.169,E2 -474.169} C_VEL
LIN {X 0,Y 608.423,Z 282.192,A -85,B 0,C 180,E1 -476.775,E2 -476.775} C_VEL
LIN {X 0,Y 608.477,Z 282.19,A -85,B 0,C 180,E1 -479.778,E2 -479.778} C_VEL
LIN {X 0,Y 608.439,Z 282.192,A -85,B 0,C 180,E1 -482.519,E2 -482.519} C_VEL
LIN {X 0,Y 608.425,Z 282.191,A -85,B 0,C 180,E1 -484.902,E2 -484.902} C_VEL
LIN {X 0,Y 608.464,Z 282.193,A -85,B 0,C 180,E1 -487.746,E2 -487.746} C_VEL
LIN {X 0,Y 608.433,Z 282.193,A -85,B 0,C 180,E1 -490.326,E2 -490.326} C_VEL
LIN {X 0,Y 608.481,Z 282.186,A -85,B 0,C 180,E1 -493.309,E2 -493.309} C_VEL
LIN {X 0,Y 608.461,Z 282.192,A -85,B 0,C 180,E1 -496.129,E2 -496.129} C_VEL
LIN {X 0,Y 608.438,Z 282.189,A -85,B 0,C 180,E1 -498.822,E2 -498.822} C_VEL
LIN {X 0,Y 608.463,Z 282.197,A -85,B 0,C 180,E1 -501.759,E2 -501.759} C_VEL
LIN {X 0,Y 608.437,Z 282.196,A -85,B 0,C 180,E1 -503.954,E2 -503.954} C_VEL
LIN {X 0,Y 608.434,Z 282.191,A -85,B 0,C 180,E1 -506.327,E2 -506.327} C_VEL
LIN {X 0,Y 608.438,Z 282.189,A -85,B 0,C 180,E1 -508.732,E2 -508.732} C_VEL
LIN {X 0,Y 608.478,Z 282.191,A -85,B 0,C 180,E1 -511.377,E2 -511.377} C_VEL
LIN {X 0,Y 608.432,Z 282.194,A -85,B 0,C 180,E1 -513.964,E2 -513.964} C_VEL
LIN {X 0,Y 608.445,Z 282.19,A -85,B 0,C 180,E1 -516.154,E2 -516.154} C_VEL
LIN {X 0,Y 608.452,Z 282.188,A -85,B 0,C 180,E1 -518.307,E2 -518.307} C_VEL
LIN {X 0,Y 608.472,Z 282.192,A -85,B 0,C 180,E1 -521.28,E2 -521.28} C_VEL
LIN {X 0,Y 608.444,Z 282.192,A -85,B 0,C 180,E1 -523.905,E2 -523.905} C_VEL
LIN {X 0,Y 608.464,Z 282.186,A -85,B 0,C 180,E1 -526.643,E2 -526.643} C_VEL
LIN {X 0,Y 608.463,Z 282.196,A -85,B 0,C 180,E1 -529.35,E2 -529.35} C_VEL
LIN {X 0,Y 608.46,Z 282.187,A -85,B 0,C 180,E1 -532.032,E2 -532.032} C_VEL
LIN {X 0,Y 608.467,Z 282.187,A -85,B 0,C 180,E1 -534.698,E2 -534.698} C_VEL
LIN {X 0,Y 608.474,Z 282.194,A -85,B 0,C 180,E1 -537.352,E2 -537.352} C_VEL
LIN {X 0,Y 608.457,Z 282.187,A -85,B 0,C 180,E1 -540,E2 -540} C_VEL
LIN {X 0,Y 608.481,Z 282.186,A -85,B 0,C 180,E1 -542.648,E2 -542.648} C_VEL
LIN {X 0,Y 608.463,Z 282.194,A -85,B 0,C 180,E1 -545.301,E2 -545.301} C_VEL
LIN {X 0,Y 608.46,Z 282.186,A -85,B 0,C 180,E1 -547.967,E2 -547.967} C_VEL
LIN {X 0,Y 608.452,Z 282.191,A -85,B 0,C 180,E1 -549.472,E2 -549.472} C_VEL
LIN {X 0,Y 607.766,Z 282.275,A -85,B 0,C 180,E1 -550.025,E2 -550.025} C_VEL
LIN {X 0,Y 604.907,Z 282.636,A -85,B 0,C 180,E1 -550.922,E2 -550.922} C_VEL
LIN {X 0,Y 602.507,Z 282.93,A -85,B 0,C 180,E1 -551.643,E2 -551.643} C_VEL
LIN {X 0,Y 601.482,Z 283.056,A -85,B 0,C 180,E1 -552.2,E2 -552.2} C_VEL
LIN {X 0,Y 601.402,Z 283.066,A -85,B 0,C 180,E1 -552.388,E2 -552.388} C_VEL
LIN {X 0,Y 601.425,Z 283.071,A -85,B 0,C 180,E1 -554.897,E2 -554.897} C_VEL
LIN {X 0,Y 601.423,Z 283.074,A -85,B 0,C 180,E1 -556.986,E2 -556.986} C_VEL
LIN {X 0,Y 601.4,Z 283.065,A -85,B 0,C 180,E1 -559.809,E2 -559.809} C_VEL
LIN {X 0,Y 601.403,Z 283.072,A -85,B 0,C 180,E1 -562.683,E2 -562.683} C_VEL
LIN {X 0,Y 601.398,Z 283.077,A -85,B 0,C 180,E1 -564.878,E2 -564.878} C_VEL
LIN {X 0,Y 601.414,Z 283.063,A -85,B 0,C 180,E1 -567.867,E2 -567.867} C_VEL
LIN {X 0,Y 601.438,Z 283.062,A -85,B 0,C 180,E1 -570.163,E2 -570.163} C_VEL
LIN {X 0,Y 601.415,Z 283.074,A -85,B 0,C 180,E1 -572.716,E2 -572.716} C_VEL
LIN {X 0,Y 601.411,Z 283.069,A -85,B 0,C 180,E1 -575.116,E2 -575.116} C_VEL
LIN {X 0,Y 601.425,Z 283.064,A -85,B 0,C 180,E1 -577.419,E2 -577.419} C_VEL
LIN {X 0,Y 601.407,Z 283.066,A -85,B 0,C 180,E1 -579.995,E2 -579.995} C_VEL
LIN {X 0,Y 601.404,Z 283.076,A -85,B 0,C 180,E1 -582.67,E2 -582.67} C_VEL
LIN {X 0,Y 601.416,Z 283.064,A -85,B 0,C 180,E1 -585.482,E2 -585.482} C_VEL
LIN {X 0,Y 601.423,Z 283.069,A -85,B 0,C 180,E1 -588.406,E2 -588.406} C_VEL
LIN {X 0,Y 601.426,Z 283.068,A -85,B 0,C 180,E1 -590.876,E2 -590.876} C_VEL
LIN {X 0,Y 601.436,Z 283.062,A -85,B 0,C 180,E1 -593.734,E2 -593.734} C_VEL
LIN {X 0,Y 601.427,Z 283.069,A -85,B 0,C 180,E1 -596.687,E2 -596.687} C_VEL
LIN {X 0,Y 601.423,Z 283.064,A -85,B 0,C 180,E1 -599.059,E2 -599.059} C_VEL
LIN {X 0,Y 601.431,Z 283.062,A -85,B 0,C 180,E1 -601.374,E2 -601.374} C_VEL
LIN {X 0,Y 601.417,Z 283.071,A -85,B 0,C 180,E1 -604.131,E2 -604.131} C_VEL
LIN {X 0,Y 601.417,Z 283.07,A -85,B 0,C 180,E1 -606.59,E2 -606.59} C_VEL
LIN {X 0,Y 601.429,Z 283.063,A -85,B 0,C 180,E1 -609.479,E2 -609.479} C_VEL
LIN {X 0,Y 601.394,Z 283.077,A -85,B 0,C 180,E1 -612.312,E2 -612.312} C_VEL
LIN {X 0,Y 601.41,Z 283.072,A -85,B 0,C 180,E1 -614.409,E2 -614.409} C_VEL
LIN {X 0,Y 601.416,Z 283.064,A -85,B 0,C 180,E1 -617.172,E2 -617.172} C_VEL
LIN {X 0,Y 601.438,Z 283.068,A -85,B 0,C 180,E1 -619.905,E2 -619.905} C_VEL
LIN {X 0,Y 601.437,Z 283.064,A -85,B 0,C 180,E1 -622.615,E2 -622.615} C_VEL
LIN {X 0,Y 601.418,Z 283.065,A -85,B 0,C 180,E1 -625.308,E2 -625.308} C_VEL
LIN {X 0,Y 601.436,Z 283.072,A -85,B 0,C 180,E1 -627.991,E2 -627.991} C_VEL
LIN {X 0,Y 601.446,Z 283.062,A -85,B 0,C 180,E1 -630.67,E2 -630.67} C_VEL
LIN {X 0,Y 601.425,Z 283.065,A -85,B 0,C 180,E1 -633.349,E2 -633.349} C_VEL
LIN {X 0,Y 601.42,Z 283.072,A -85,B 0,C 180,E1 -636.037,E2 -636.037} C_VEL
LIN {X 0,Y 601.411,Z 283.065,A -85,B 0,C 180,E1 -638.738,E2 -638.738} C_VEL
LIN {X 0,Y 601.431,Z 283.067,A -85,B 0,C 180,E1 -641.458,E2 -641.458} C_VEL
LIN {X 0,Y 601.416,Z 283.068,A -85,B 0,C 180,E1 -644.205,E2 -644.205} C_VEL
LIN {X 0,Y 601.429,Z 283.063,A -85,B 0,C 180,E1 -646.986,E2 -646.986} C_VEL
LIN {X 0,Y 601.401,Z 283.075,A -85,B 0,C 180,E1 -649.809,E2 -649.809} C_VEL
LIN {X 0,Y 601.41,Z 283.065,A -85,B 0,C 180,E1 -652.605,E2 -652.605} C_VEL
LIN {X 0,Y 601.398,Z 283.067,A -85,B 0,C 180,E1 -654.878,E2 -654.878} C_VEL
LIN {X 0,Y 601.418,Z 283.07,A -85,B 0,C 180,E1 -657.867,E2 -657.867} C_VEL
LIN {X 0,Y 601.422,Z 283.065,A -85,B 0,C 180,E1 -660.164,E2 -660.164} C_VEL
LIN {X 0,Y 601.423,Z 283.063,A -85,B 0,C 180,E1 -662.716,E2 -662.716} C_VEL
LIN {X 0,Y 601.405,Z 283.068,A -85,B 0,C 180,E1 -665.114,E2 -665.114} C_VEL
LIN {X 0,Y 601.428,Z 283.072,A -85,B 0,C 180,E1 -667.419,E2 -667.419} C_VEL
LIN {X 0,Y 601.405,Z 283.067,A -85,B 0,C 180,E1 -669.994,E2 -669.994} C_VEL
LIN {X 0,Y 601.407,Z 283.064,A -85,B 0,C 180,E1 -672.669,E2 -672.669} C_VEL
LIN {X 0,Y 601.416,Z 283.073,A -85,B 0,C 180,E1 -675.482,E2 -675.482} C_VEL
LIN {X 0,Y 601.416,Z 283.064,A -85,B 0,C 180,E1 -678.406,E2 -678.406} C_VEL
LIN {X 0,Y 601.426,Z 283.066,A -85,B 0,C 180,E1 -680.875,E2 -680.875} C_VEL
LIN {X 0,Y 601.436,Z 283.064,A -85,B 0,C 180,E1 -683.733,E2 -683.733} C_VEL
LIN {X 0,Y 601.425,Z 283.063,A -85,B 0,C 180,E1 -686.063,E2 -686.063} C_VEL
LIN {X 0,Y 601.431,Z 283.063,A -85,B 0,C 180,E1 -688.541,E2 -688.541} C_VEL
LIN {X 0,Y 601.43,Z 283.068,A -85,B 0,C 180,E1 -691.374,E2 -691.374} C_VEL
LIN {X 0,Y 601.397,Z 283.069,A -85,B 0,C 180,E1 -693.636,E2 -693.636} C_VEL
LIN {X 0,Y 601.414,Z 283.067,A -85,B 0,C 180,E1 -696.59,E2 -696.59} C_VEL
LIN {X 0,Y 601.429,Z 283.065,A -85,B 0,C 180,E1 -699.479,E2 -699.479} C_VEL
LIN {X 0,Y 601.388,Z 283.068,A -85,B 0,C 180,E1 -702.312,E2 -702.312} C_VEL
LIN {X 0,Y 601.407,Z 283.067,A -85,B 0,C 180,E1 -704.409,E2 -704.409} C_VEL
LIN {X 0,Y 601.42,Z 283.07,A -85,B 0,C 180,E1 -707.172,E2 -707.172} C_VEL
LIN {X 0,Y 601.422,Z 283.062,A -85,B 0,C 180,E1 -709.905,E2 -709.905} C_VEL
LIN {X 0,Y 601.444,Z 283.066,A -85,B 0,C 180,E1 -712.615,E2 -712.615} C_VEL
LIN {X 0,Y 601.425,Z 283.066,A -85,B 0,C 180,E1 -715.308,E2 -715.308} C_VEL
LIN {X 0,Y 601.408,Z 283.065,A -85,B 0,C 180,E1 -717.991,E2 -717.991} C_VEL
LIN {X 0,Y 601.451,Z 283.067,A -85,B 0,C 180,E1 -720.67,E2 -720.67} C_VEL
LIN {X 0,Y 601.429,Z 283.064,A -85,B 0,C 180,E1 -723.35,E2 -723.35} C_VEL
LIN {X 0,Y 601.395,Z 283.068,A -85,B 0,C 180,E1 -726.038,E2 -726.038} C_VEL
LIN {X 0,Y 601.436,Z 283.069,A -85,B 0,C 180,E1 -728.738,E2 -728.738} C_VEL
LIN {X 0,Y 601.426,Z 283.062,A -85,B 0,C 180,E1 -731.459,E2 -731.459} C_VEL
LIN {X 0,Y 601.41,Z 283.069,A -85,B 0,C 180,E1 -734.206,E2 -734.206} C_VEL
LIN {X 0,Y 601.428,Z 283.065,A -85,B 0,C 180,E1 -736.986,E2 -736.986} C_VEL
LIN {X 0,Y 601.397,Z 283.066,A -85,B 0,C 180,E1 -739.81,E2 -739.81} C_VEL
LIN {X 0,Y 601.409,Z 283.073,A -85,B 0,C 180,E1 -742.607,E2 -742.607} C_VEL
LIN {X 0,Y 601.397,Z 283.069,A -85,B 0,C 180,E1 -744.879,E2 -744.879} C_VEL
LIN {X 0,Y 601.414,Z 283.066,A -85,B 0,C 180,E1 -747.868,E2 -747.868} C_VEL
LIN {X 0,Y 601.419,Z 283.071,A -85,B 0,C 180,E1 -750.165,E2 -750.165} C_VEL
LIN {X 0,Y 601.422,Z 283.067,A -85,B 0,C 180,E1 -752.718,E2 -752.718} C_VEL
LIN {X 0,Y 601.406,Z 283.065,A -85,B 0,C 180,E1 -755.115,E2 -755.115} C_VEL
LIN {X 0,Y 601.427,Z 283.063,A -85,B 0,C 180,E1 -757.42,E2 -757.42} C_VEL
LIN {X 0,Y 601.397,Z 283.073,A -85,B 0,C 180,E1 -759.997,E2 -759.997} C_VEL
LIN {X 0,Y 601.408,Z 283.068,A -85,B 0,C 180,E1 -762.671,E2 -762.671} C_VEL
LIN {X 0,Y 601.393,Z 283.068,A -85,B 0,C 180,E1 -765.48,E2 -765.48} C_VEL
LIN {X 0,Y 601.381,Z 283.069,A -85,B 0,C 180,E1 -767.413,E2 -767.413} C_VEL
LIN {X 0,Y 601.399,Z 283.074,A -85,B 0,C 180,E1 -770.005,E2 -770.005} C_VEL
LIN {X 0,Y 601.431,Z 283.064,A -85,B 0,C 180,E1 -772.619,E2 -772.619} C_VEL
LIN {X 0,Y 601.389,Z 283.067,A -85,B 0,C 180,E1 -775.067,E2 -775.067} C_VEL
LIN {X 0,Y 601.41,Z 283.067,A -85,B 0,C 180,E1 -777.484,E2 -777.484} C_VEL
LIN {X 0,Y 601.428,Z 283.072,A -85,B 0,C 180,E1 -779.852,E2 -779.852} C_VEL
LIN {X 0,Y 601.413,Z 283.065,A -85,B 0,C 180,E1 -782.888,E2 -782.888} C_VEL
LIN {X 0,Y 601.457,Z 283.216,A -85,B 0,C 180,E1 -785.704,E2 -785.704} C_VEL
LIN {X 0,Y 601.571,Z 292.531,A -85,B 0,C 180,E1 -787.36,E2 -787.36} C_VEL
LIN {X 0,Y 601.559,Z 307.848,A -85,B 0,C 180,E1 -790.018,E2 -790.018} C_VEL
LIN {X 0,Y 601.496,Z 325.439,A -85,B 0,C 180,E1 -793.016,E2 -793.016} C_VEL
LIN {X 0,Y 601.425,Z 342.673,A -85,B 0,C 180,E1 -795.908,E2 -795.908} C_VEL
LIN {X 0,Y 601.462,Z 348.245,A -85,B 0,C 180,E1 -796.808,E2 -796.808} C_VEL
LIN {X 0,Y 601.687,Z 350.746,A -85,B 0,C 180,E1 -796.877,E2 -796.877} C_VEL
LIN {X 0,Y 601.62,Z 454.913,A -85,B 0,C 180,E1 -798.14,E2 -798.14} C_VEL
LIN {X 0,Y 601.59,Z 468.244,A -85,B 0,C 180,E1 -798.438,E2 -798.438} C_VEL
LIN {X 0,Y 601.548,Z 480.667,A -85,B 0,C 180,E1 -798.854,E2 -798.854} C_VEL
LIN {X 0,Y 601.519,Z 492.61,A -85,B 0,C 180,E1 -799.396,E2 -799.396} C_VEL
LIN {X 0,Y 601.487,Z 504.203,A -85,B 0,C 180,E1 -800.076,E2 -800.076} C_VEL
LIN {X 0,Y 601.438,Z 515.647,A -85,B 0,C 180,E1 -800.924,E2 -800.924} C_VEL
LIN {X 0,Y 601.411,Z 524.778,A -85,B 0,C 180,E1 -801.77,E2 -801.77} C_VEL
LIN {X 0,Y 601.388,Z 533.683,A -85,B 0,C 180,E1 -802.783,E2 -802.783} C_VEL
LIN {X 0,Y 601.375,Z 540.774,A -85,B 0,C 180,E1 -803.782,E2 -803.782} C_VEL
LIN {X 0,Y 601.345,Z 547.365,A -85,B 0,C 180,E1 -804.971,E2 -804.971} C_VEL
LIN {X 0,Y 601.346,Z 551.672,A -85,B 0,C 180,E1 -805.979,E2 -805.979} C_VEL
LIN {X 0,Y 601.344,Z 553.959,A -85,B 0,C 180,E1 -806.65,E2 -806.65} C_VEL
LIN {X 0,Y 601.325,Z 555.804,A -85,B 0,C 180,E1 -807.321,E2 -807.321} C_VEL
LIN {X 0,Y 601.343,Z 557.199,A -85,B 0,C 180,E1 -807.991,E2 -807.991} C_VEL
LIN {X 0,Y 601.339,Z 558.783,A -85,B 0,C 180,E1 -809.33,E2 -809.33} C_VEL
LIN {X 0,Y 601.335,Z 558.99,A -85,B 0,C 180,E1 -810,E2 -810} C_VEL
LIN {X 0,Y 601.348,Z 558.186,A -85,B 0,C 180,E1 -811.339,E2 -811.339} C_VEL
LIN {X 0,Y 601.343,Z 557.199,A -85,B 0,C 180,E1 -812.009,E2 -812.009} C_VEL
LIN {X 0,Y 601.325,Z 555.804,A -85,B 0,C 180,E1 -812.679,E2 -812.679} C_VEL
LIN {X 0,Y 601.367,Z 552.894,A -85,B 0,C 180,E1 -813.685,E2 -813.685} C_VEL
LIN {X 0,Y 601.336,Z 548.949,A -85,B 0,C 180,E1 -814.693,E2 -814.693} C_VEL
LIN {X 0,Y 601.374,Z 543.856,A -85,B 0,C 180,E1 -815.701,E2 -815.701} C_VEL
LIN {X 0,Y 601.382,Z 537.47,A -85,B 0,C 180,E1 -816.711,E2 -816.711} C_VEL
LIN {X 0,Y 601.396,Z 529.484,A -85,B 0,C 180,E1 -817.723,E2 -817.723} C_VEL
LIN {X 0,Y 601.423,Z 521.343,A -85,B 0,C 180,E1 -818.568,E2 -818.568} C_VEL
LIN {X 0,Y 601.451,Z 511.386,A -85,B 0,C 180,E1 -819.415,E2 -819.415} C_VEL
LIN {X 0,Y 601.48,Z 501.572,A -85,B 0,C 180,E1 -820.094,E2 -820.094} C_VEL
LIN {X 0,Y 601.529,Z 490.934,A -85,B 0,C 180,E1 -820.689,E2 -820.689} C_VEL
LIN {X 0,Y 601.572,Z 477.571,A -85,B 0,C 180,E1 -821.263,E2 -821.263} C_VEL
LIN {X 0,Y 601.593,Z 465.047,A -85,B 0,C 180,E1 -821.647,E2 -821.647} C_VEL
LIN {X 0,Y 601.637,Z 452.128,A -85,B 0,C 180,E1 -821.902,E2 -821.902} C_VEL
LIN {X 0,Y 601.548,Z 349.242,A -85,B 0,C 180,E1 -823.147,E2 -823.147} C_VEL
LIN {X 0,Y 601.457,Z 348.03,A -85,B 0,C 180,E1 -823.214,E2 -823.214} C_VEL
LIN {X 0,Y 601.469,Z 330.613,A -85,B 0,C 180,E1 -826.111,E2 -826.111} C_VEL
LIN {X 0,Y 601.525,Z 314.464,A -85,B 0,C 180,E1 -828.848,E2 -828.848} C_VEL
LIN {X 0,Y 601.565,Z 298.535,A -85,B 0,C 180,E1 -831.592,E2 -831.592} C_VEL
LIN {X 0,Y 601.582,Z 284.048,A -85,B 0,C 180,E1 -834.134,E2 -834.134} C_VEL
LIN {X 0,Y 601.419,Z 283.087,A -85,B 0,C 180,E1 -834.383,E2 -834.383} C_VEL
LIN {X 0,Y 601.413,Z 283.065,A -85,B 0,C 180,E1 -837.112,E2 -837.112} C_VEL
LIN {X 0,Y 601.428,Z 283.072,A -85,B 0,C 180,E1 -840.148,E2 -840.148} C_VEL
LIN {X 0,Y 601.405,Z 283.066,A -85,B 0,C 180,E1 -842.712,E2 -842.712} C_VEL
LIN {X 0,Y 601.383,Z 283.068,A -85,B 0,C 180,E1 -845.11,E2 -845.11} C_VEL
LIN {X 0,Y 601.43,Z 283.065,A -85,B 0,C 180,E1 -847.418,E2 -847.418} C_VEL
LIN {X 0,Y 601.399,Z 283.074,A -85,B 0,C 180,E1 -849.995,E2 -849.995} C_VEL
LIN {X 0,Y 601.382,Z 283.069,A -85,B 0,C 180,E1 -852.672,E2 -852.672} C_VEL
LIN {X 0,Y 601.392,Z 283.068,A -85,B 0,C 180,E1 -854.532,E2 -854.532} C_VEL
LIN {X 0,Y 601.411,Z 283.069,A -85,B 0,C 180,E1 -857.408,E2 -857.408} C_VEL
LIN {X 0,Y 601.397,Z 283.072,A -85,B 0,C 180,E1 -860.003,E2 -860.003} C_VEL
LIN {X 0,Y 601.428,Z 283.063,A -85,B 0,C 180,E1 -862.617,E2 -862.617} C_VEL
LIN {X 0,Y 601.435,Z 283.063,A -85,B 0,C 180,E1 -865.069,E2 -865.069} C_VEL
LIN {X 0,Y 601.434,Z 283.068,A -85,B 0,C 180,E1 -867.484,E2 -867.484} C_VEL
LIN {X 0,Y 601.419,Z 283.07,A -85,B 0,C 180,E1 -869.851,E2 -869.851} C_VEL
LIN {X 0,Y 601.414,Z 283.066,A -85,B 0,C 180,E1 -872.132,E2 -872.132} C_VEL
LIN {X 0,Y 601.397,Z 283.069,A -85,B 0,C 180,E1 -875.121,E2 -875.121} C_VEL
LIN {X 0,Y 601.409,Z 283.073,A -85,B 0,C 180,E1 -877.393,E2 -877.393} C_VEL
LIN {X 0,Y 601.397,Z 283.066,A -85,B 0,C 180,E1 -880.19,E2 -880.19} C_VEL
LIN {X 0,Y 601.428,Z 283.065,A -85,B 0,C 180,E1 -883.014,E2 -883.014} C_VEL
LIN {X 0,Y 601.41,Z 283.067,A -85,B 0,C 180,E1 -885.907,E2 -885.907} C_VEL
LIN {X 0,Y 601.428,Z 283.062,A -85,B 0,C 180,E1 -888.541,E2 -888.541} C_VEL
LIN {X 0,Y 601.436,Z 283.069,A -85,B 0,C 180,E1 -891.262,E2 -891.262} C_VEL
LIN {X 0,Y 601.395,Z 283.068,A -85,B 0,C 180,E1 -893.962,E2 -893.962} C_VEL
LIN {X 0,Y 601.429,Z 283.064,A -85,B 0,C 180,E1 -896.65,E2 -896.65} C_VEL
LIN {X 0,Y 601.451,Z 283.067,A -85,B 0,C 180,E1 -899.33,E2 -899.33} C_VEL
LIN {X 0,Y 601.408,Z 283.065,A -85,B 0,C 180,E1 -902.009,E2 -902.009} C_VEL
LIN {X 0,Y 601.427,Z 283.066,A -85,B 0,C 180,E1 -904.692,E2 -904.692} C_VEL
LIN {X 0,Y 601.444,Z 283.066,A -85,B 0,C 180,E1 -907.385,E2 -907.385} C_VEL
LIN {X 0,Y 601.422,Z 283.062,A -85,B 0,C 180,E1 -910.095,E2 -910.095} C_VEL
LIN {X 0,Y 601.402,Z 283.066,A -85,B 0,C 180,E1 -912.388,E2 -912.388} C_VEL
LIN {X 0,Y 600.743,Z 283.156,A -85,B 0,C 180,E1 -912.948,E2 -912.948} C_VEL
LIN {X 0,Y 597.893,Z 283.515,A -85,B 0,C 180,E1 -913.856,E2 -913.856} C_VEL
LIN {X 0,Y 595.479,Z 283.816,A -85,B 0,C 180,E1 -914.586,E2 -914.586} C_VEL
LIN {X 0,Y 594.44,Z 283.941,A -85,B 0,C 180,E1 -915.149,E2 -915.149} C_VEL
LIN {X 0,Y 594.354,Z 283.949,A -85,B 0,C 180,E1 -915.34,E2 -915.34} C_VEL
LIN {X 0,Y 594.38,Z 283.946,A -85,B 0,C 180,E1 -917.193,E2 -917.193} C_VEL
LIN {X 0,Y 594.37,Z 283.94,A -85,B 0,C 180,E1 -920.053,E2 -920.053} C_VEL
LIN {X 0,Y 594.355,Z 283.953,A -85,B 0,C 180,E1 -922.967,E2 -922.967} C_VEL
LIN {X 0,Y 594.367,Z 283.947,A -85,B 0,C 180,E1 -925.193,E2 -925.193} C_VEL
LIN {X 0,Y 594.374,Z 283.941,A -85,B 0,C 180,E1 -927.527,E2 -927.527} C_VEL
LIN {X 0,Y 594.391,Z 283.942,A -85,B 0,C 180,E1 -930.331,E2 -930.331} C_VEL
LIN {X 0,Y 594.369,Z 283.949,A -85,B 0,C 180,E1 -932.95,E2 -932.95} C_VEL
LIN {X 0,Y 594.376,Z 283.942,A -85,B 0,C 180,E1 -935.407,E2 -935.407} C_VEL
LIN {X 0,Y 594.381,Z 283.941,A -85,B 0,C 180,E1 -937.941,E2 -937.941} C_VEL
LIN {X 0,Y 594.378,Z 283.948,A -85,B 0,C 180,E1 -940.824,E2 -940.824} C_VEL
LIN {X 0,Y 594.373,Z 283.942,A -85,B 0,C 180,E1 -943.841,E2 -943.841} C_VEL
LIN {X 0,Y 594.372,Z 283.947,A -85,B 0,C 180,E1 -946.702,E2 -946.702} C_VEL
LIN {X 0,Y 594.366,Z 283.941,A -85,B 0,C 180,E1 -949.434,E2 -949.434} C_VEL
LIN {X 0,Y 594.383,Z 283.949,A -85,B 0,C 180,E1 -952.392,E2 -952.392} C_VEL
LIN {X 0,Y 594.377,Z 283.946,A -85,B 0,C 180,E1 -954.672,E2 -954.672} C_VEL
LIN {X 0,Y 594.375,Z 283.943,A -85,B 0,C 180,E1 -957.088,E2 -957.088} C_VEL
LIN {X 0,Y 594.381,Z 283.941,A -85,B 0,C 180,E1 -959.672,E2 -959.672} C_VEL
LIN {X 0,Y 594.368,Z 283.95,A -85,B 0,C 180,E1 -962.539,E2 -962.539} C_VEL
LIN {X 0,Y 594.374,Z 283.945,A -85,B 0,C 180,E1 -964.808,E2 -964.808} C_VEL
LIN {X 0,Y 594.36,Z 283.943,A -85,B 0,C 180,E1 -967.265,E2 -967.265} C_VEL
LIN {X 0,Y 594.372,Z 283.947,A -85,B 0,C 180,E1 -969.947,E2 -969.947} C_VEL
LIN {X 0,Y 594.386,Z 283.942,A -85,B 0,C 180,E1 -972.807,E2 -972.807} C_VEL
LIN {X 0,Y 594.385,Z 283.945,A -85,B 0,C 180,E1 -975.826,E2 -975.826} C_VEL
LIN {X 0,Y 594.39,Z 283.946,A -85,B 0,C 180,E1 -978.404,E2 -978.404} C_VEL
LIN {X 0,Y 594.378,Z 283.941,A -85,B 0,C 180,E1 -981.158,E2 -981.158} C_VEL
LIN {X 0,Y 594.375,Z 283.949,A -85,B 0,C 180,E1 -983.891,E2 -983.891} C_VEL
LIN {X 0,Y 594.377,Z 283.943,A -85,B 0,C 180,E1 -986.611,E2 -986.611} C_VEL
LIN {X 0,Y 594.417,Z 283.937,A -85,B 0,C 180,E1 -989.323,E2 -989.323} C_VEL
LIN {X 0,Y 594.404,Z 283.948,A -85,B 0,C 180,E1 -992.033,E2 -992.033} C_VEL
LIN {X 0,Y 594.387,Z 283.94,A -85,B 0,C 180,E1 -994.748,E2 -994.748} C_VEL
LIN {X 0,Y 594.39,Z 283.943,A -85,B 0,C 180,E1 -997.473,E2 -997.473} C_VEL
LIN {X 0,Y 594.396,Z 283.943,A -85,B 0,C 180,E1 -1000.216,E2 -1000.216} C_VEL
LIN {X 0,Y 594.363,Z 283.943,A -85,B 0,C 180,E1 -1002.983,E2 -1002.983} C_VEL
LIN {X 0,Y 594.364,Z 283.953,A -85,B 0,C 180,E1 -1005.781,E2 -1005.781} C_VEL
LIN {X 0,Y 594.384,Z 283.94,A -85,B 0,C 180,E1 -1008.617,E2 -1008.617} C_VEL
LIN {X 0,Y 594.363,Z 283.95,A -85,B 0,C 180,E1 -1011.503,E2 -1011.503} C_VEL
LIN {X 0,Y 594.383,Z 283.941,A -85,B 0,C 180,E1 -1014.446,E2 -1014.446} C_VEL
LIN {X 0,Y 594.38,Z 283.941,A -85,B 0,C 180,E1 -1016.699,E2 -1016.699} C_VEL
LIN {X 0,Y 594.378,Z 283.942,A -85,B 0,C 180,E1 -1018.998,E2 -1018.998} C_VEL
LIN {X 0,Y 594.389,Z 283.949,A -85,B 0,C 180,E1 -1021.645,E2 -1021.645} C_VEL
LIN {X 0,Y 594.386,Z 283.938,A -85,B 0,C 180,E1 -1024.579,E2 -1024.579} C_VEL
LIN {X 0,Y 594.378,Z 283.944,A -85,B 0,C 180,E1 -1027.086,E2 -1027.086} C_VEL
LIN {X 0,Y 594.369,Z 283.946,A -85,B 0,C 180,E1 -1029.774,E2 -1029.774} C_VEL
LIN {X 0,Y 594.366,Z 283.94,A -85,B 0,C 180,E1 -1032.374,E2 -1032.374} C_VEL
LIN {X 0,Y 594.354,Z 283.95,A -85,B 0,C 180,E1 -1035.191,E2 -1035.191} C_VEL
LIN {X 0,Y 594.362,Z 283.948,A -85,B 0,C 180,E1 -1037.625,E2 -1037.625} C_VEL
LIN {X 0,Y 594.385,Z 283.939,A -85,B 0,C 180,E1 -1040.321,E2 -1040.321} C_VEL
LIN {X 0,Y 594.376,Z 283.945,A -85,B 0,C 180,E1 -1042.913,E2 -1042.913} C_VEL
LIN {X 0,Y 594.379,Z 283.941,A -85,B 0,C 180,E1 -1045.86,E2 -1045.86} C_VEL
LIN {X 0,Y 594.381,Z 283.943,A -85,B 0,C 180,E1 -1048.651,E2 -1048.651} C_VEL
LIN {X 0,Y 594.377,Z 283.949,A -85,B 0,C 180,E1 -1051.041,E2 -1051.041} C_VEL
LIN {X 0,Y 594.376,Z 283.941,A -85,B 0,C 180,E1 -1053.977,E2 -1053.977} C_VEL
LIN {X 0,Y 594.387,Z 283.94,A -85,B 0,C 180,E1 -1056.296,E2 -1056.296} C_VEL
LIN {X 0,Y 594.399,Z 283.944,A -85,B 0,C 180,E1 -1059.225,E2 -1059.225} C_VEL
LIN {X 0,Y 594.37,Z 283.941,A -85,B 0,C 180,E1 -1062.096,E2 -1062.096} C_VEL
LIN {X 0,Y 594.361,Z 283.943,A -85,B 0,C 180,E1 -1064.219,E2 -1064.219} C_VEL
LIN {X 0,Y 594.365,Z 283.951,A -85,B 0,C 180,E1 -1067.017,E2 -1067.017} C_VEL
LIN {X 0,Y 594.384,Z 283.938,A -85,B 0,C 180,E1 -1069.784,E2 -1069.784} C_VEL
LIN {X 0,Y 594.392,Z 283.943,A -85,B 0,C 180,E1 -1072.527,E2 -1072.527} C_VEL
LIN {X 0,Y 594.393,Z 283.942,A -85,B 0,C 180,E1 -1075.253,E2 -1075.253} C_VEL
LIN {X 0,Y 594.379,Z 283.94,A -85,B 0,C 180,E1 -1077.968,E2 -1077.968} C_VEL
LIN {X 0,Y 594.421,Z 283.942,A -85,B 0,C 180,E1 -1080.678,E2 -1080.678} C_VEL
LIN {X 0,Y 594.379,Z 283.942,A -85,B 0,C 180,E1 -1083.39,E2 -1083.39} C_VEL
LIN {X 0,Y 594.352,Z 283.946,A -85,B 0,C 180,E1 -1086.109,E2 -1086.109} C_VEL
LIN {X 0,Y 594.396,Z 283.943,A -85,B 0,C 180,E1 -1088.842,E2 -1088.842} C_VEL
LIN {X 0,Y 594.384,Z 283.939,A -85,B 0,C 180,E1 -1091.596,E2 -1091.596} C_VEL
LIN {X 0,Y 594.381,Z 283.947,A -85,B 0,C 180,E1 -1094.378,E2 -1094.378} C_VEL
LIN {X 0,Y 594.383,Z 283.94,A -85,B 0,C 180,E1 -1097.194,E2 -1097.194} C_VEL
LIN {X 0,Y 594.369,Z 283.944,A -85,B 0,C 180,E1 -1100.054,E2 -1100.054} C_VEL
LIN {X 0,Y 594.355,Z 283.946,A -85,B 0,C 180,E1 -1102.968,E2 -1102.968} C_VEL
LIN {X 0,Y 594.364,Z 283.942,A -85,B 0,C 180,E1 -1105.194,E2 -1105.194} C_VEL
LIN {X 0,Y 594.377,Z 283.94,A -85,B 0,C 180,E1 -1107.528,E2 -1107.528} C_VEL
LIN {X 0,Y 594.377,Z 283.951,A -85,B 0,C 180,E1 -1110.329,E2 -1110.329} C_VEL
LIN {X 0,Y 594.372,Z 283.942,A -85,B 0,C 180,E1 -1112.951,E2 -1112.951} C_VEL
LIN {X 0,Y 594.348,Z 283.944,A -85,B 0,C 180,E1 -1115.41,E2 -1115.41} C_VEL
LIN {X 0,Y 594.381,Z 283.945,A -85,B 0,C 180,E1 -1117.941,E2 -1117.941} C_VEL
LIN {X 0,Y 594.37,Z 283.943,A -85,B 0,C 180,E1 -1120.823,E2 -1120.823} C_VEL
LIN {X 0,Y 594.361,Z 283.943,A -85,B 0,C 180,E1 -1123.3,E2 -1123.3} C_VEL
LIN {X 0,Y 594.372,Z 283.952,A -85,B 0,C 180,E1 -1126.161,E2 -1126.161} C_VEL
LIN {X 0,Y 594.369,Z 283.94,A -85,B 0,C 180,E1 -1129.179,E2 -1129.179} C_VEL
LIN {X 0,Y 594.378,Z 283.951,A -85,B 0,C 180,E1 -1132.06,E2 -1132.06} C_VEL
LIN {X 0,Y 594.346,Z 283.946,A -85,B 0,C 180,E1 -1134.678,E2 -1134.678} C_VEL
LIN {X 0,Y 594.374,Z 283.941,A -85,B 0,C 180,E1 -1137.09,E2 -1137.09} C_VEL
LIN {X 0,Y 594.384,Z 283.946,A -85,B 0,C 180,E1 -1139.673,E2 -1139.673} C_VEL
LIN {X 0,Y 594.375,Z 283.944,A -85,B 0,C 180,E1 -1142.54,E2 -1142.54} C_VEL
LIN {X 0,Y 594.389,Z 284.024,A -85,B 0,C 180,E1 -1145.531,E2 -1145.531} C_VEL
LIN {X 0,Y 594.665,Z 288.187,A -85,B 0,C 180,E1 -1146.308,E2 -1146.308} C_VEL
LIN {X 0,Y 594.563,Z 304.743,A -85,B 0,C 180,E1 -1149.231,E2 -1149.231} C_VEL
LIN {X 0,Y 594.487,Z 320.265,A -85,B 0,C 180,E1 -1151.922,E2 -1151.922} C_VEL
LIN {X 0,Y 594.441,Z 335.786,A -85,B 0,C 180,E1 -1154.573,E2 -1154.573} C_VEL
LIN {X 0,Y 594.426,Z 348.24,A -85,B 0,C 180,E1 -1156.649,E2 -1156.649} C_VEL
LIN {X 0,Y 594.77,Z 350.746,A -85,B 0,C 180,E1 -1156.722,E2 -1156.722} C_VEL
LIN {X 0,Y 594.672,Z 454.857,A -85,B 0,C 180,E1 -1157.999,E2 -1157.999} C_VEL
LIN {X 0,Y 594.638,Z 468.253,A -85,B 0,C 180,E1 -1158.301,E2 -1158.301} C_VEL
LIN {X 0,Y 594.593,Z 481.339,A -85,B 0,C 180,E1 -1158.748,E2 -1158.748} C_VEL
LIN {X 0,Y 594.536,Z 492.592,A -85,B 0,C 180,E1 -1159.27,E2 -1159.27} C_VEL
LIN {X 0,Y 594.458,Z 502.905,A -85,B 0,C 180,E1 -1159.872,E2 -1159.872} C_VEL
LIN {X 0,Y 594.404,Z 513.545,A -85,B 0,C 180,E1 -1160.644,E2 -1160.644} C_VEL
LIN {X 0,Y 594.383,Z 523.121,A -85,B 0,C 180,E1 -1161.501,E2 -1161.501} C_VEL
LIN {X 0,Y 594.347,Z 530.949,A -85,B 0,C 180,E1 -1162.356,E2 -1162.356} C_VEL
LIN {X 0,Y 594.303,Z 538.693,A -85,B 0,C 180,E1 -1163.391,E2 -1163.391} C_VEL
LIN {X 0,Y 594.289,Z 545.682,A -85,B 0,C 180,E1 -1164.571,E2 -1164.571} C_VEL
LIN {X 0,Y 594.27,Z 550.376,A -85,B 0,C 180,E1 -1165.591,E2 -1165.591} C_VEL
LIN {X 0,Y 594.267,Z 553.962,A -85,B 0,C 180,E1 -1166.61,E2 -1166.61} C_VEL
LIN {X 0,Y 594.225,Z 555.799,A -85,B 0,C 180,E1 -1167.288,E2 -1167.288} C_VEL
LIN {X 0,Y 594.242,Z 557.192,A -85,B 0,C 180,E1 -1167.967,E2 -1167.967} C_VEL
LIN {X 0,Y 594.248,Z 558.187,A -85,B 0,C 180,E1 -1168.645,E2 -1168.645} C_VEL
LIN {X 0,Y 594.239,Z 558.782,A -85,B 0,C 180,E1 -1169.322,E2 -1169.322} C_VEL
LIN {X 0,Y 594.236,Z 558.982,A -85,B 0,C 180,E1 -1170,E2 -1170} C_VEL
LIN {X 0,Y 594.239,Z 558.782,A -85,B 0,C 180,E1 -1170.678,E2 -1170.678} C_VEL
LIN {X 0,Y 594.248,Z 558.187,A -85,B 0,C 180,E1 -1171.355,E2 -1171.355} C_VEL
LIN {X 0,Y 594.242,Z 557.192,A -85,B 0,C 180,E1 -1172.033,E2 -1172.033} C_VEL
LIN {X 0,Y 594.225,Z 555.799,A -85,B 0,C 180,E1 -1172.712,E2 -1172.712} C_VEL
LIN {X 0,Y 594.288,Z 552.889,A -85,B 0,C 180,E1 -1173.729,E2 -1173.729} C_VEL
LIN {X 0,Y 594.241,Z 548.941,A -85,B 0,C 180,E1 -1174.749,E2 -1174.749} C_VEL
LIN {X 0,Y 594.3,Z 543.847,A -85,B 0,C 180,E1 -1175.769,E2 -1175.769} C_VEL
LIN {X 0,Y 594.316,Z 537.463,A -85,B 0,C 180,E1 -1176.791,E2 -1176.791} C_VEL
LIN {X 0,Y 594.346,Z 529.487,A -85,B 0,C 180,E1 -1177.815,E2 -1177.815} C_VEL
LIN {X 0,Y 594.377,Z 521.347,A -85,B 0,C 180,E1 -1178.671,E2 -1178.671} C_VEL
LIN {X 0,Y 594.414,Z 511.372,A -85,B 0,C 180,E1 -1179.528,E2 -1179.528} C_VEL
LIN {X 0,Y 594.468,Z 501.556,A -85,B 0,C 180,E1 -1180.214,E2 -1180.214} C_VEL
LIN {X 0,Y 594.55,Z 490.938,A -85,B 0,C 180,E1 -1180.816,E2 -1180.816} C_VEL
LIN {X 0,Y 594.598,Z 478.055,A -85,B 0,C 180,E1 -1181.379,E2 -1181.379} C_VEL
LIN {X 0,Y 594.654,Z 465.887,A -85,B 0,C 180,E1 -1181.763,E2 -1181.763} C_VEL
LIN {X 0,Y 594.678,Z 453.526,A -85,B 0,C 180,E1 -1182.022,E2 -1182.022} C_VEL
LIN {X 0,Y 594.668,Z 350.077,A -85,B 0,C 180,E1 -1183.288,E2 -1183.288} C_VEL
LIN {X 0,Y 594.426,Z 348.241,A -85,B 0,C 180,E1 -1183.351,E2 -1183.351} C_VEL
LIN {X 0,Y 594.459,Z 331.647,A -85,B 0,C 180,E1 -1186.13,E2 -1186.13} C_VEL
LIN {X 0,Y 594.53,Z 315.094,A -85,B 0,C 180,E1 -1188.969,E2 -1188.969} C_VEL
LIN {X 0,Y 594.604,Z 300.604,A -85,B 0,C 180,E1 -1191.494,E2 -1191.494} C_VEL
LIN {X 0,Y 594.673,Z 286.145,A -85,B 0,C 180,E1 -1194.057,E2 -1194.057} C_VEL
LIN {X 0,Y 594.383,Z 283.98,A -85,B 0,C 180,E1 -1194.492,E2 -1194.492} C_VEL
LIN {X 0,Y 594.375,Z 283.944,A -85,B 0,C 180,E1 -1197.46,E2 -1197.46} C_VEL
LIN {X 0,Y 594.384,Z 283.946,A -85,B 0,C 180,E1 -1200.327,E2 -1200.327} C_VEL
LIN {X 0,Y 594.374,Z 283.941,A -85,B 0,C 180,E1 -1202.95,E2 -1202.95} C_VEL
LIN {X 0,Y 594.345,Z 283.947,A -85,B 0,C 180,E1 -1205.408,E2 -1205.408} C_VEL
LIN {X 0,Y 594.378,Z 283.951,A -85,B 0,C 180,E1 -1207.94,E2 -1207.94} C_VEL
LIN {X 0,Y 594.369,Z 283.94,A -85,B 0,C 180,E1 -1210.821,E2 -1210.821} C_VEL
LIN {X 0,Y 594.372,Z 283.952,A -85,B 0,C 180,E1 -1213.839,E2 -1213.839} C_VEL
LIN {X 0,Y 594.361,Z 283.943,A -85,B 0,C 180,E1 -1216.7,E2 -1216.7} C_VEL
LIN {X 0,Y 594.382,Z 283.945,A -85,B 0,C 180,E1 -1219.434,E2 -1219.434} C_VEL
LIN {X 0,Y 594.383,Z 283.941,A -85,B 0,C 180,E1 -1222.391,E2 -1222.391} C_VEL
LIN {X 0,Y 594.388,Z 283.945,A -85,B 0,C 180,E1 -1225.42,E2 -1225.42} C_VEL
LIN {X 0,Y 594.37,Z 283.943,A -85,B 0,C 180,E1 -1228.356,E2 -1228.356} C_VEL
LIN {X 0,Y 594.378,Z 283.942,A -85,B 0,C 180,E1 -1231.041,E2 -1231.041} C_VEL
LIN {X 0,Y 594.371,Z 283.945,A -85,B 0,C 180,E1 -1233.978,E2 -1233.978} C_VEL
LIN {X 0,Y 594.377,Z 283.941,A -85,B 0,C 180,E1 -1236.295,E2 -1236.295} C_VEL
LIN {X 0,Y 594.403,Z 283.943,A -85,B 0,C 180,E1 -1239.224,E2 -1239.224} C_VEL
LIN {X 0,Y 594.346,Z 283.945,A -85,B 0,C 180,E1 -1242.094,E2 -1242.094} C_VEL
LIN {X 0,Y 594.359,Z 283.943,A -85,B 0,C 180,E1 -1244.219,E2 -1244.219} C_VEL
LIN {X 0,Y 594.369,Z 283.946,A -85,B 0,C 180,E1 -1247.017,E2 -1247.017} C_VEL
LIN {X 0,Y 594.381,Z 283.942,A -85,B 0,C 180,E1 -1249.784,E2 -1249.784} C_VEL
LIN {X 0,Y 594.393,Z 283.938,A -85,B 0,C 180,E1 -1252.526,E2 -1252.526} C_VEL
LIN {X 0,Y 594.392,Z 283.949,A -85,B 0,C 180,E1 -1255.252,E2 -1255.252} C_VEL
LIN {X 0,Y 594.378,Z 283.941,A -85,B 0,C 180,E1 -1257.967,E2 -1257.967} C_VEL
LIN {X 0,Y 594.42,Z 283.935,A -85,B 0,C 180,E1 -1260.677,E2 -1260.677} C_VEL
LIN {X 0,Y 594.379,Z 283.947,A -85,B 0,C 180,E1 -1263.389,E2 -1263.389} C_VEL
LIN {X 0,Y 594.353,Z 283.944,A -85,B 0,C 180,E1 -1266.109,E2 -1266.109} C_VEL
LIN {X 0,Y 594.394,Z 283.944,A -85,B 0,C 180,E1 -1268.842,E2 -1268.842} C_VEL
LIN {X 0,Y 594.384,Z 283.942,A -85,B 0,C 180,E1 -1271.595,E2 -1271.595} C_VEL
LIN {X 0,Y 594.379,Z 283.942,A -85,B 0,C 180,E1 -1274.377,E2 -1274.377} C_VEL
LIN {X 0,Y 594.354,Z 283.949,A -85,B 0,C 180,E1 -1275.34,E2 -1275.34} C_VEL
LIN {X 0,Y 593.68,Z 284.03,A -85,B 0,C 180,E1 -1275.906,E2 -1275.906} C_VEL
LIN {X 0,Y 590.813,Z 284.392,A -85,B 0,C 180,E1 -1276.824,E2 -1276.824} C_VEL
LIN {X 0,Y 588.402,Z 284.687,A -85,B 0,C 180,E1 -1277.563,E2 -1277.563} C_VEL
LIN {X 0,Y 587.379,Z 284.812,A -85,B 0,C 180,E1 -1278.133,E2 -1278.133} C_VEL
LIN {X 0,Y 587.303,Z 284.822,A -85,B 0,C 180,E1 -1278.326,E2 -1278.326} C_VEL
LIN {X 0,Y 587.347,Z 284.825,A -85,B 0,C 180,E1 -1281.045,E2 -1281.045} C_VEL
LIN {X 0,Y 587.33,Z 284.819,A -85,B 0,C 180,E1 -1284.006,E2 -1284.006} C_VEL
LIN {X 0,Y 587.329,Z 284.82,A -85,B 0,C 180,E1 -1286.279,E2 -1286.279} C_VEL
LIN {X 0,Y 587.343,Z 284.822,A -85,B 0,C 180,E1 -1289.135,E2 -1289.135} C_VEL
LIN {X 0,Y 587.346,Z 284.817,A -85,B 0,C 180,E1 -1291.838,E2 -1291.838} C_VEL
LIN {X 0,Y 587.35,Z 284.819,A -85,B 0,C 180,E1 -1294.35,E2 -1294.35} C_VEL
LIN {X 0,Y 587.344,Z 284.828,A -85,B 0,C 180,E1 -1296.747,E2 -1296.747} C_VEL
LIN {X 0,Y 587.339,Z 284.818,A -85,B 0,C 180,E1 -1299.359,E2 -1299.359} C_VEL
LIN {X 0,Y 587.325,Z 284.821,A -85,B 0,C 180,E1 -1302.108,E2 -1302.108} C_VEL
LIN {X 0,Y 587.307,Z 284.824,A -85,B 0,C 180,E1 -1305.089,E2 -1305.089} C_VEL
LIN {X 0,Y 587.344,Z 284.815,A -85,B 0,C 180,E1 -1307.928,E2 -1307.928} C_VEL
LIN {X 0,Y 587.326,Z 284.822,A -85,B 0,C 180,E1 -1311.058,E2 -1311.058} C_VEL
LIN {X 0,Y 587.346,Z 284.817,A -85,B 0,C 180,E1 -1313.292,E2 -1313.292} C_VEL
LIN {X 0,Y 587.36,Z 284.813,A -85,B 0,C 180,E1 -1315.781,E2 -1315.781} C_VEL
LIN {X 0,Y 587.35,Z 284.823,A -85,B 0,C 180,E1 -1318.232,E2 -1318.232} C_VEL
LIN {X 0,Y 587.345,Z 284.819,A -85,B 0,C 180,E1 -1320.866,E2 -1320.866} C_VEL
LIN {X 0,Y 587.358,Z 284.818,A -85,B 0,C 180,E1 -1323.818,E2 -1323.818} C_VEL
LIN {X 0,Y 587.333,Z 284.824,A -85,B 0,C 180,E1 -1325.994,E2 -1325.994} C_VEL
LIN {X 0,Y 587.318,Z 284.83,A -85,B 0,C 180,E1 -1328.226,E2 -1328.226} C_VEL
LIN {X 0,Y 587.347,Z 284.817,A -85,B 0,C 180,E1 -1331.152,E2 -1331.152} C_VEL
LIN {X 0,Y 587.348,Z 284.817,A -85,B 0,C 180,E1 -1333.311,E2 -1333.311} C_VEL
LIN {X 0,Y 587.356,Z 284.826,A -85,B 0,C 180,E1 -1336.155,E2 -1336.155} C_VEL
LIN {X 0,Y 587.34,Z 284.818,A -85,B 0,C 180,E1 -1338.963,E2 -1338.963} C_VEL
LIN {X 0,Y 587.363,Z 284.82,A -85,B 0,C 180,E1 -1341.745,E2 -1341.745} C_VEL
LIN {X 0,Y 587.356,Z 284.82,A -85,B 0,C 180,E1 -1344.507,E2 -1344.507} C_VEL
LIN {X 0,Y 587.369,Z 284.815,A -85,B 0,C 180,E1 -1347.257,E2 -1347.257} C_VEL
LIN {X 0,Y 587.382,Z 284.823,A -85,B 0,C 180,E1 -1350,E2 -1350} C_VEL
LIN {X 0,Y 587.369,Z 284.815,A -85,B 0,C 180,E1 -1352.743,E2 -1352.743} C_VEL
LIN {X 0,Y 587.356,Z 284.82,A -85,B 0,C 180,E1 -1355.493,E2 -1355.493} C_VEL
LIN {X 0,Y 587.363,Z 284.82,A -85,B 0,C 180,E1 -1358.255,E2 -1358.255} C_VEL
LIN {X 0,Y 587.344,Z 284.818,A -85,B 0,C 180,E1 -1361.133,E2 -1361.133} C_VEL
LIN {X 0,Y 587.361,Z 284.819,A -85,B 0,C 180,E1 -1364.26,E2 -1364.26} C_VEL
LIN {X 0,Y 587.354,Z 284.821,A -85,B 0,C 180,E1 -1367.405,E2 -1367.405} C_VEL
LIN {X 0,Y 587.327,Z 284.822,A -85,B 0,C 180,E1 -1370.304,E2 -1370.304} C_VEL
LIN {X 0,Y 587.318,Z 284.824,A -85,B 0,C 180,E1 -1373.258,E2 -1373.258} C_VEL
LIN {X 0,Y 587.335,Z 284.827,A -85,B 0,C 180,E1 -1375.516,E2 -1375.516} C_VEL
LIN {X 0,Y 587.344,Z 284.823,A -85,B 0,C 180,E1 -1377.817,E2 -1377.817} C_VEL
LIN {X 0,Y 587.335,Z 284.818,A -85,B 0,C 180,E1 -1380.51,E2 -1380.51} C_VEL
LIN {X 0,Y 587.335,Z 284.822,A -85,B 0,C 180,E1 -1383.112,E2 -1383.112} C_VEL
LIN {X 0,Y 587.349,Z 284.82,A -85,B 0,C 180,E1 -1385.895,E2 -1385.895} C_VEL
LIN {X 0,Y 587.325,Z 284.819,A -85,B 0,C 180,E1 -1388.479,E2 -1388.479} C_VEL
LIN {X 0,Y 587.331,Z 284.823,A -85,B 0,C 180,E1 -1391.156,E2 -1391.156} C_VEL
LIN {X 0,Y 587.325,Z 284.819,A -85,B 0,C 180,E1 -1394.114,E2 -1394.114} C_VEL
LIN {X 0,Y 587.312,Z 284.825,A -85,B 0,C 180,E1 -1396.994,E2 -1396.994} C_VEL
LIN {X 0,Y 587.319,Z 284.823,A -85,B 0,C 180,E1 -1399.747,E2 -1399.747} C_VEL
LIN {X 0,Y 587.336,Z 284.818,A -85,B 0,C 180,E1 -1402.392,E2 -1402.392} C_VEL
LIN {X 0,Y 587.343,Z 284.822,A -85,B 0,C 180,E1 -1404.946,E2 -1404.946} C_VEL
LIN {X 0,Y 587.331,Z 284.826,A -85,B 0,C 180,E1 -1407.421,E2 -1407.421} C_VEL
LIN {X 0,Y 587.337,Z 284.819,A -85,B 0,C 180,E1 -1409.831,E2 -1409.831} C_VEL
LIN {X 0,Y 587.341,Z 284.816,A -85,B 0,C 180,E1 -1412.307,E2 -1412.307} C_VEL
LIN {X 0,Y 587.325,Z 284.82,A -85,B 0,C 180,E1 -1414.483,E2 -1414.483} C_VEL
LIN {X 0,Y 587.31,Z 284.831,A -85,B 0,C 180,E1 -1417.13,E2 -1417.13} C_VEL
LIN {X 0,Y 587.325,Z 284.819,A -85,B 0,C 180,E1 -1419.695,E2 -1419.695} C_VEL
LIN {X 0,Y 587.347,Z 284.819,A -85,B 0,C 180,E1 -1422.594,E2 -1422.594} C_VEL
LIN {X 0,Y 587.353,Z 284.816,A -85,B 0,C 180,E1 -1425.739,E2 -1425.739} C_VEL
LIN {X 0,Y 587.351,Z 284.825,A -85,B 0,C 180,E1 -1428.859,E2 -1428.859} C_VEL
LIN {X 0,Y 587.359,Z 284.814,A -85,B 0,C 180,E1 -1431.745,E2 -1431.745} C_VEL
LIN {X 0,Y 587.351,Z 284.821,A -85,B 0,C 180,E1 -1434.507,E2 -1434.507} C_VEL
LIN {X 0,Y 587.375,Z 284.815,A -85,B 0,C 180,E1 -1437.257,E2 -1437.257} C_VEL
LIN {X 0,Y 587.365,Z 284.812,A -85,B 0,C 180,E1 -1440,E2 -1440} C_VEL
LIN {X 0,Y 587.37,Z 284.824,A -85,B 0,C 180,E1 -1442.744,E2 -1442.744} C_VEL
LIN {X 0,Y 587.353,Z 284.816,A -85,B 0,C 180,E1 -1445.493,E2 -1445.493} C_VEL
LIN {X 0,Y 587.36,Z 284.818,A -85,B 0,C 180,E1 -1448.256,E2 -1448.256} C_VEL
LIN {X 0,Y 587.353,Z 284.817,A -85,B 0,C 180,E1 -1451.142,E2 -1451.142} C_VEL
LIN {X 0,Y 587.354,Z 284.82,A -85,B 0,C 180,E1 -1454.261,E2 -1454.261} C_VEL
LIN {X 0,Y 587.343,Z 284.815,A -85,B 0,C 180,E1 -1457.407,E2 -1457.407} C_VEL
LIN {X 0,Y 587.326,Z 284.824,A -85,B 0,C 180,E1 -1460.305,E2 -1460.305} C_VEL
LIN {X 0,Y 587.312,Z 284.821,A -85,B 0,C 180,E1 -1463.259,E2 -1463.259} C_VEL
LIN {X 0,Y 587.321,Z 284.819,A -85,B 0,C 180,E1 -1465.518,E2 -1465.518} C_VEL
LIN {X 0,Y 587.343,Z 284.817,A -85,B 0,C 180,E1 -1467.818,E2 -1467.818} C_VEL
LIN {X 0,Y 587.329,Z 284.827,A -85,B 0,C 180,E1 -1470.511,E2 -1470.511} C_VEL
LIN {X 0,Y 587.321,Z 284.819,A -85,B 0,C 180,E1 -1473.398,E2 -1473.398} C_VEL
LIN {X 0,Y 587.287,Z 284.828,A -85,B 0,C 180,E1 -1475.901,E2 -1475.901} C_VEL
LIN {X 0,Y 587.324,Z 284.825,A -85,B 0,C 180,E1 -1478.48,E2 -1478.48} C_VEL
LIN {X 0,Y 587.329,Z 284.819,A -85,B 0,C 180,E1 -1481.158,E2 -1481.158} C_VEL
LIN {X 0,Y 587.322,Z 284.829,A -85,B 0,C 180,E1 -1484.114,E2 -1484.114} C_VEL
LIN {X 0,Y 587.303,Z 284.822,A -85,B 0,C 180,E1 -1486.994,E2 -1486.994} C_VEL
LIN {X 0,Y 587.306,Z 284.824,A -85,B 0,C 180,E1 -1489.746,E2 -1489.746} C_VEL
LIN {X 0,Y 587.34,Z 284.822,A -85,B 0,C 180,E1 -1492.393,E2 -1492.393} C_VEL
LIN {X 0,Y 587.355,Z 284.822,A -85,B 0,C 180,E1 -1495.78,E2 -1495.78} C_VEL
LIN {X 0,Y 587.336,Z 284.825,A -85,B 0,C 180,E1 -1498.232,E2 -1498.232} C_VEL
LIN {X 0,Y 587.344,Z 284.818,A -85,B 0,C 180,E1 -1500.868,E2 -1500.868} C_VEL
LIN {X 0,Y 587.327,Z 284.828,A -85,B 0,C 180,E1 -1503.722,E2 -1503.722} C_VEL
LIN {X 0,Y 587.37,Z 284.947,A -85,B 0,C 180,E1 -1505.389,E2 -1505.389} C_VEL
LIN {X 0,Y 587.741,Z 289.222,A -85,B 0,C 180,E1 -1506.199,E2 -1506.199} C_VEL
LIN {X 0,Y 587.598,Z 305.778,A -85,B 0,C 180,E1 -1509.156,E2 -1509.156} C_VEL
LIN {X 0,Y 587.494,Z 322.334,A -85,B 0,C 180,E1 -1512.059,E2 -1512.059} C_VEL
LIN {X 0,Y 587.4,Z 338.891,A -85,B 0,C 180,E1 -1514.917,E2 -1514.917} C_VEL
LIN {X 0,Y 587.395,Z 348.236,A -85,B 0,C 180,E1 -1516.486,E2 -1516.486} C_VEL
LIN {X 0,Y 587.764,Z 350.746,A -85,B 0,C 180,E1 -1516.561,E2 -1516.561} C_VEL
LIN {X 0,Y 587.734,Z 454.801,A -85,B 0,C 180,E1 -1517.856,E2 -1517.856} C_VEL
LIN {X 0,Y 587.693,Z 467.504,A -85,B 0,C 180,E1 -1518.139,E2 -1518.139} C_VEL
LIN {X 0,Y 587.609,Z 480.828,A -85,B 0,C 180,E1 -1518.592,E2 -1518.592} C_VEL
LIN {X 0,Y 587.555,Z 492.574,A -85,B 0,C 180,E1 -1519.141,E2 -1519.141} C_VEL
LIN {X 0,Y 587.442,Z 502.888,A -85,B 0,C 180,E1 -1519.749,E2 -1519.749} C_VEL
LIN {X 0,Y 587.378,Z 513.549,A -85,B 0,C 180,E1 -1520.531,E2 -1520.531} C_VEL
LIN {X 0,Y 587.322,Z 523.122,A -85,B 0,C 180,E1 -1521.398,E2 -1521.398} C_VEL
LIN {X 0,Y 587.273,Z 530.94,A -85,B 0,C 180,E1 -1522.263,E2 -1522.263} C_VEL
LIN {X 0,Y 587.229,Z 537.454,A -85,B 0,C 180,E1 -1523.126,E2 -1523.126} C_VEL
LIN {X 0,Y 587.23,Z 543.837,A -85,B 0,C 180,E1 -1524.161,E2 -1524.161} C_VEL
LIN {X 0,Y 587.146,Z 548.933,A -85,B 0,C 180,E1 -1525.194,E2 -1525.194} C_VEL
LIN {X 0,Y 587.212,Z 552.882,A -85,B 0,C 180,E1 -1526.226,E2 -1526.226} C_VEL
LIN {X 0,Y 587.132,Z 555.794,A -85,B 0,C 180,E1 -1527.256,E2 -1527.256} C_VEL
LIN {X 0,Y 587.147,Z 558.189,A -85,B 0,C 180,E1 -1528.628,E2 -1528.628} C_VEL
LIN {X 0,Y 587.14,Z 558.782,A -85,B 0,C 180,E1 -1529.314,E2 -1529.314} C_VEL
LIN {X 0,Y 587.14,Z 558.782,A -85,B 0,C 180,E1 -1530.686,E2 -1530.686} C_VEL
LIN {X 0,Y 587.147,Z 558.189,A -85,B 0,C 180,E1 -1531.372,E2 -1531.372} C_VEL
LIN {X 0,Y 587.132,Z 555.794,A -85,B 0,C 180,E1 -1532.744,E2 -1532.744} C_VEL
LIN {X 0,Y 587.212,Z 552.882,A -85,B 0,C 180,E1 -1533.774,E2 -1533.774} C_VEL
LIN {X 0,Y 587.146,Z 548.933,A -85,B 0,C 180,E1 -1534.806,E2 -1534.806} C_VEL
LIN {X 0,Y 587.23,Z 543.837,A -85,B 0,C 180,E1 -1535.839,E2 -1535.839} C_VEL
LIN {X 0,Y 587.229,Z 537.454,A -85,B 0,C 180,E1 -1536.874,E2 -1536.874} C_VEL
LIN {X 0,Y 587.287,Z 529.491,A -85,B 0,C 180,E1 -1537.91,E2 -1537.91} C_VEL
LIN {X 0,Y 587.335,Z 521.35,A -85,B 0,C 180,E1 -1538.775,E2 -1538.775} C_VEL
LIN {X 0,Y 587.386,Z 511.359,A -85,B 0,C 180,E1 -1539.643,E2 -1539.643} C_VEL
LIN {X 0,Y 587.467,Z 501.54,A -85,B 0,C 180,E1 -1540.337,E2 -1540.337} C_VEL
LIN {X 0,Y 587.552,Z 490.938,A -85,B 0,C 180,E1 -1540.946,E2 -1540.946} C_VEL
LIN {X 0,Y 587.616,Z 477.245,A -85,B 0,C 180,E1 -1541.547,E2 -1541.547} C_VEL
LIN {X 0,Y 587.689,Z 464.98,A -85,B 0,C 180,E1 -1541.926,E2 -1541.926} C_VEL
LIN {X 0,Y 587.737,Z 453.47,A -85,B 0,C 180,E1 -1542.166,E2 -1542.166} C_VEL
LIN {X 0,Y 587.764,Z 350.746,A -85,B 0,C 180,E1 -1543.439,E2 -1543.439} C_VEL
LIN {X 0,Y 587.395,Z 348.237,A -85,B 0,C 180,E1 -1543.514,E2 -1543.514} C_VEL
LIN {X 0,Y 587.44,Z 331.647,A -85,B 0,C 180,E1 -1546.328,E2 -1546.328} C_VEL
LIN {X 0,Y 587.546,Z 315.708,A -85,B 0,C 180,E1 -1549.096,E2 -1549.096} C_VEL
LIN {X 0,Y 587.63,Z 300.604,A -85,B 0,C 180,E1 -1551.762,E2 -1551.762} C_VEL
LIN {X 0,Y 587.758,Z 288.187,A -85,B 0,C 180,E1 -1553.988,E2 -1553.988} C_VEL
LIN {X 0,Y 587.359,Z 284.907,A -85,B 0,C 180,E1 -1554.629,E2 -1554.629} C_VEL
LIN {X 0,Y 587.34,Z 284.823,A -85,B 0,C 180,E1 -1557.69,E2 -1557.69} C_VEL
LIN {X 0,Y 587.333,Z 284.822,A -85,B 0,C 180,E1 -1560.509,E2 -1560.509} C_VEL
LIN {X 0,Y 587.333,Z 284.82,A -85,B 0,C 180,E1 -1563.396,E2 -1563.396} C_VEL
LIN {X 0,Y 587.287,Z 284.833,A -85,B 0,C 180,E1 -1565.899,E2 -1565.899} C_VEL
LIN {X 0,Y 587.317,Z 284.822,A -85,B 0,C 180,E1 -1568.479,E2 -1568.479} C_VEL
LIN {X 0,Y 587.332,Z 284.817,A -85,B 0,C 180,E1 -1571.156,E2 -1571.156} C_VEL
LIN {X 0,Y 587.316,Z 284.826,A -85,B 0,C 180,E1 -1574.112,E2 -1574.112} C_VEL
LIN {X 0,Y 587.31,Z 284.822,A -85,B 0,C 180,E1 -1576.993,E2 -1576.993} C_VEL
LIN {X 0,Y 587.316,Z 284.83,A -85,B 0,C 180,E1 -1579.745,E2 -1579.745} C_VEL
LIN {X 0,Y 587.338,Z 284.819,A -85,B 0,C 180,E1 -1582.391,E2 -1582.391} C_VEL
LIN {X 0,Y 587.344,Z 284.826,A -85,B 0,C 180,E1 -1585.651,E2 -1585.651} C_VEL
LIN {X 0,Y 587.335,Z 284.82,A -85,B 0,C 180,E1 -1588.23,E2 -1588.23} C_VEL
LIN {X 0,Y 587.342,Z 284.818,A -85,B 0,C 180,E1 -1590.866,E2 -1590.866} C_VEL
LIN {X 0,Y 587.348,Z 284.822,A -85,B 0,C 180,E1 -1593.819,E2 -1593.819} C_VEL
LIN {X 0,Y 587.325,Z 284.822,A -85,B 0,C 180,E1 -1595.993,E2 -1595.993} C_VEL
LIN {X 0,Y 587.34,Z 284.819,A -85,B 0,C 180,E1 -1598.962,E2 -1598.962} C_VEL
LIN {X 0,Y 587.346,Z 284.82,A -85,B 0,C 180,E1 -1601.151,E2 -1601.151} C_VEL
LIN {X 0,Y 587.316,Z 284.822,A -85,B 0,C 180,E1 -1604.024,E2 -1604.024} C_VEL
LIN {X 0,Y 587.35,Z 284.817,A -85,B 0,C 180,E1 -1606.154,E2 -1606.154} C_VEL
LIN {X 0,Y 587.338,Z 284.82,A -85,B 0,C 180,E1 -1608.962,E2 -1608.962} C_VEL
LIN {X 0,Y 587.36,Z 284.818,A -85,B 0,C 180,E1 -1611.744,E2 -1611.744} C_VEL
LIN {X 0,Y 587.353,Z 284.816,A -85,B 0,C 180,E1 -1614.507,E2 -1614.507} C_VEL
LIN {X 0,Y 587.37,Z 284.824,A -85,B 0,C 180,E1 -1617.256,E2 -1617.256} C_VEL
LIN {X 0,Y 587.365,Z 284.812,A -85,B 0,C 180,E1 -1620,E2 -1620} C_VEL
LIN {X 0,Y 587.375,Z 284.815,A -85,B 0,C 180,E1 -1622.743,E2 -1622.743} C_VEL
LIN {X 0,Y 587.351,Z 284.821,A -85,B 0,C 180,E1 -1625.493,E2 -1625.493} C_VEL
LIN {X 0,Y 587.359,Z 284.814,A -85,B 0,C 180,E1 -1628.255,E2 -1628.255} C_VEL
LIN {X 0,Y 587.351,Z 284.825,A -85,B 0,C 180,E1 -1631.141,E2 -1631.141} C_VEL
LIN {X 0,Y 587.353,Z 284.816,A -85,B 0,C 180,E1 -1634.261,E2 -1634.261} C_VEL
LIN {X 0,Y 587.34,Z 284.82,A -85,B 0,C 180,E1 -1637.406,E2 -1637.406} C_VEL
LIN {X 0,Y 587.303,Z 284.822,A -85,B 0,C 180,E1 -1638.326,E2 -1638.326} C_VEL
LIN {X 0,Y 586.661,Z 284.91,A -85,B 0,C 180,E1 -1638.898,E2 -1638.898} C_VEL
LIN {X 0,Y 583.836,Z 285.264,A -85,B 0,C 180,E1 -1639.827,E2 -1639.827} C_VEL
LIN {X 0,Y 581.425,Z 285.564,A -85,B 0,C 180,E1 -1640.574,E2 -1640.574} C_VEL
LIN {X 0,Y 580.371,Z 285.692,A -85,B 0,C 180,E1 -1641.15,E2 -1641.15} C_VEL
LIN {X 0,Y 580.276,Z 285.701,A -85,B 0,C 180,E1 -1641.345,E2 -1641.345} C_VEL
LIN {X 0,Y 580.291,Z 285.697,A -85,B 0,C 180,E1 -1644.316,E2 -1644.316} C_VEL
LIN {X 0,Y 580.268,Z 285.704,A -85,B 0,C 180,E1 -1646.623,E2 -1646.623} C_VEL
LIN {X 0,Y 580.297,Z 285.698,A -85,B 0,C 180,E1 -1649.311,E2 -1649.311} C_VEL
LIN {X 0,Y 580.293,Z 285.697,A -85,B 0,C 180,E1 -1652.2,E2 -1652.2} C_VEL
LIN {X 0,Y 580.294,Z 285.703,A -85,B 0,C 180,E1 -1654.695,E2 -1654.695} C_VEL
LIN {X 0,Y 580.291,Z 285.698,A -85,B 0,C 180,E1 -1657.268,E2 -1657.268} C_VEL
LIN {X 0,Y 580.297,Z 285.698,A -85,B 0,C 180,E1 -1660.273,E2 -1660.273} C_VEL
LIN {X 0,Y 580.272,Z 285.707,A -85,B 0,C 180,E1 -1662.706,E2 -1662.706} C_VEL
LIN {X 0,Y 580.265,Z 285.698,A -85,B 0,C 180,E1 -1665.609,E2 -1665.609} C_VEL
LIN {X 0,Y 580.306,Z 285.694,A -85,B 0,C 180,E1 -1668.235,E2 -1668.235} C_VEL
LIN {X 0,Y 580.281,Z 285.7,A -85,B 0,C 180,E1 -1670.966,E2 -1670.966} C_VEL
LIN {X 0,Y 580.289,Z 285.696,A -85,B 0,C 180,E1 -1673.599,E2 -1673.599} C_VEL
LIN {X 0,Y 580.314,Z 285.695,A -85,B 0,C 180,E1 -1676.146,E2 -1676.146} C_VEL
LIN {X 0,Y 580.284,Z 285.703,A -85,B 0,C 180,E1 -1678.616,E2 -1678.616} C_VEL
LIN {X 0,Y 580.289,Z 285.697,A -85,B 0,C 180,E1 -1681.024,E2 -1681.024} C_VEL
LIN {X 0,Y 580.323,Z 285.693,A -85,B 0,C 180,E1 -1683.659,E2 -1683.659} C_VEL
LIN {X 0,Y 580.275,Z 285.706,A -85,B 0,C 180,E1 -1686.442,E2 -1686.442} C_VEL
LIN {X 0,Y 580.271,Z 285.699,A -85,B 0,C 180,E1 -1689.438,E2 -1689.438} C_VEL
LIN {X 0,Y 580.276,Z 285.7,A -85,B 0,C 180,E1 -1691.646,E2 -1691.646} C_VEL
LIN {X 0,Y 580.276,Z 285.702,A -85,B 0,C 180,E1 -1693.826,E2 -1693.826} C_VEL
LIN {X 0,Y 580.322,Z 285.699,A -85,B 0,C 180,E1 -1695.983,E2 -1695.983} C_VEL
LIN {X 0,Y 580.301,Z 285.696,A -85,B 0,C 180,E1 -1698.827,E2 -1698.827} C_VEL
LIN {X 0,Y 580.326,Z 285.695,A -85,B 0,C 180,E1 -1701.644,E2 -1701.644} C_VEL
LIN {X 0,Y 580.323,Z 285.697,A -85,B 0,C 180,E1 -1704.44,E2 -1704.44} C_VEL
LIN {X 0,Y 580.335,Z 285.691,A -85,B 0,C 180,E1 -1707.224,E2 -1707.224} C_VEL
LIN {X 0,Y 580.351,Z 285.699,A -85,B 0,C 180,E1 -1710,E2 -1710} C_VEL
LIN {X 0,Y 580.335,Z 285.691,A -85,B 0,C 180,E1 -1712.776,E2 -1712.776} C_VEL
LIN {X 0,Y 580.323,Z 285.697,A -85,B 0,C 180,E1 -1715.56,E2 -1715.56} C_VEL
LIN {X 0,Y 580.326,Z 285.695,A -85,B 0,C 180,E1 -1718.356,E2 -1718.356} C_VEL
LIN {X 0,Y 580.296,Z 285.697,A -85,B 0,C 180,E1 -1721.191,E2 -1721.191} C_VEL
LIN {X 0,Y 580.322,Z 285.699,A -85,B 0,C 180,E1 -1724.017,E2 -1724.017} C_VEL
LIN {X 0,Y 580.308,Z 285.694,A -85,B 0,C 180,E1 -1726.914,E2 -1726.914} C_VEL
LIN {X 0,Y 580.301,Z 285.704,A -85,B 0,C 180,E1 -1729.822,E2 -1729.822} C_VEL
LIN {X 0,Y 580.29,Z 285.696,A -85,B 0,C 180,E1 -1732.802,E2 -1732.802} C_VEL
LIN {X 0,Y 580.304,Z 285.696,A -85,B 0,C 180,E1 -1735.079,E2 -1735.079} C_VEL
LIN {X 0,Y 580.315,Z 285.698,A -85,B 0,C 180,E1 -1737.863,E2 -1737.863} C_VEL
LIN {X 0,Y 580.286,Z 285.696,A -85,B 0,C 180,E1 -1740.696,E2 -1740.696} C_VEL
LIN {X 0,Y 580.3,Z 285.701,A -85,B 0,C 180,E1 -1743.317,E2 -1743.317} C_VEL
LIN {X 0,Y 580.319,Z 285.698,A -85,B 0,C 180,E1 -1745.767,E2 -1745.767} C_VEL
LIN {X 0,Y 580.282,Z 285.698,A -85,B 0,C 180,E1 -1748.146,E2 -1748.146} C_VEL
LIN {X 0,Y 580.293,Z 285.695,A -85,B 0,C 180,E1 -1750.843,E2 -1750.843} C_VEL
LIN {X 0,Y 580.279,Z 285.702,A -85,B 0,C 180,E1 -1753.656,E2 -1753.656} C_VEL
LIN {X 0,Y 580.276,Z 285.698,A -85,B 0,C 180,E1 -1756.608,E2 -1756.608} C_VEL
LIN {X 0,Y 580.295,Z 285.702,A -85,B 0,C 180,E1 -1759.157,E2 -1759.157} C_VEL
LIN {X 0,Y 580.282,Z 285.698,A -85,B 0,C 180,E1 -1761.926,E2 -1761.926} C_VEL
LIN {X 0,Y 580.299,Z 285.694,A -85,B 0,C 180,E1 -1764.457,E2 -1764.457} C_VEL
LIN {X 0,Y 580.282,Z 285.702,A -85,B 0,C 180,E1 -1766.975,E2 -1766.975} C_VEL
LIN {X 0,Y 580.301,Z 285.7,A -85,B 0,C 180,E1 -1769.426,E2 -1769.426} C_VEL
LIN {X 0,Y 580.31,Z 285.691,A -85,B 0,C 180,E1 -1772.137,E2 -1772.137} C_VEL
LIN {X 0,Y 580.311,Z 285.701,A -85,B 0,C 180,E1 -1775.269,E2 -1775.269} C_VEL
LIN {X 0,Y 580.264,Z 285.699,A -85,B 0,C 180,E1 -1777.948,E2 -1777.948} C_VEL
LIN {X 0,Y 580.307,Z 285.7,A -85,B 0,C 180,E1 -1780.914,E2 -1780.914} C_VEL
LIN {X 0,Y 580.273,Z 285.698,A -85,B 0,C 180,E1 -1783.826,E2 -1783.826} C_VEL
LIN {X 0,Y 580.271,Z 285.704,A -85,B 0,C 180,E1 -1786.696,E2 -1786.696} C_VEL
LIN {X 0,Y 580.295,Z 285.693,A -85,B 0,C 180,E1 -1789.534,E2 -1789.534} C_VEL
LIN {X 0,Y 580.322,Z 285.693,A -85,B 0,C 180,E1 -1792.345,E2 -1792.345} C_VEL
LIN {X 0,Y 580.332,Z 285.696,A -85,B 0,C 180,E1 -1795.137,E2 -1795.137} C_VEL
LIN {X 0,Y 580.322,Z 285.69,A -85,B 0,C 180,E1 -1797.918,E2 -1797.918} C_VEL
LIN {X 0,Y 580.361,Z 285.692,A -85,B 0,C 180,E1 -1800.694,E2 -1800.694} C_VEL
LIN {X 0,Y 580.281,Z 285.697,A -85,B 0,C 180,E1 -1803.472,E2 -1803.472} C_VEL
LIN {X 0,Y 580.317,Z 285.692,A -85,B 0,C 180,E1 -1805.56,E2 -1805.56} C_VEL
LIN {X 0,Y 580.324,Z 285.695,A -85,B 0,C 180,E1 -1808.357,E2 -1808.357} C_VEL
LIN {X 0,Y 580.324,Z 285.692,A -85,B 0,C 180,E1 -1811.209,E2 -1811.209} C_VEL
LIN {X 0,Y 580.305,Z 285.7,A -85,B 0,C 180,E1 -1814.339,E2 -1814.339} C_VEL
LIN {X 0,Y 580.302,Z 285.696,A -85,B 0,C 180,E1 -1816.914,E2 -1816.914} C_VEL
LIN {X 0,Y 580.299,Z 285.693,A -85,B 0,C 180,E1 -1819.823,E2 -1819.823} C_VEL
LIN {X 0,Y 580.263,Z 285.702,A -85,B 0,C 180,E1 -1822.053,E2 -1822.053} C_VEL
LIN {X 0,Y 580.296,Z 285.695,A -85,B 0,C 180,E1 -1825.081,E2 -1825.081} C_VEL
LIN {X 0,Y 580.296,Z 285.7,A -85,B 0,C 180,E1 -1828.186,E2 -1828.186} C_VEL
LIN {X 0,Y 580.276,Z 285.702,A -85,B 0,C 180,E1 -1830.695,E2 -1830.695} C_VEL
LIN {X 0,Y 580.277,Z 285.696,A -85,B 0,C 180,E1 -1833.314,E2 -1833.314} C_VEL
LIN {X 0,Y 580.242,Z 285.703,A -85,B 0,C 180,E1 -1835.758,E2 -1835.758} C_VEL
LIN {X 0,Y 580.283,Z 285.705,A -85,B 0,C 180,E1 -1838.147,E2 -1838.147} C_VEL
LIN {X 0,Y 580.292,Z 285.697,A -85,B 0,C 180,E1 -1840.844,E2 -1840.844} C_VEL
LIN {X 0,Y 580.274,Z 285.7,A -85,B 0,C 180,E1 -1843.659,E2 -1843.659} C_VEL
LIN {X 0,Y 580.272,Z 285.701,A -85,B 0,C 180,E1 -1846.61,E2 -1846.61} C_VEL
LIN {X 0,Y 580.293,Z 285.693,A -85,B 0,C 180,E1 -1849.157,E2 -1849.157} C_VEL
LIN {X 0,Y 580.284,Z 285.704,A -85,B 0,C 180,E1 -1851.928,E2 -1851.928} C_VEL
LIN {X 0,Y 580.248,Z 285.705,A -85,B 0,C 180,E1 -1854.453,E2 -1854.453} C_VEL
LIN {X 0,Y 580.287,Z 285.696,A -85,B 0,C 180,E1 -1856.976,E2 -1856.976} C_VEL
LIN {X 0,Y 580.292,Z 285.699,A -85,B 0,C 180,E1 -1859.426,E2 -1859.426} C_VEL
LIN {X 0,Y 580.288,Z 285.705,A -85,B 0,C 180,E1 -1862.144,E2 -1862.144} C_VEL
LIN {X 0,Y 580.294,Z 285.756,A -85,B 0,C 180,E1 -1865.214,E2 -1865.214} C_VEL
LIN {X 0,Y 580.777,Z 289.13,A -85,B 0,C 180,E1 -1865.896,E2 -1865.896} C_VEL
LIN {X 0,Y 580.646,Z 304.959,A -85,B 0,C 180,E1 -1868.748,E2 -1868.748} C_VEL
LIN {X 0,Y 580.518,Z 319.23,A -85,B 0,C 180,E1 -1871.288,E2 -1871.288} C_VEL
LIN {X 0,Y 580.408,Z 334.752,A -85,B 0,C 180,E1 -1874.01,E2 -1874.01} C_VEL
LIN {X 0,Y 580.364,Z 348.243,A -85,B 0,C 180,E1 -1876.319,E2 -1876.319} C_VEL
LIN {X 0,Y 580.687,Z 350.746,A -85,B 0,C 180,E1 -1876.394,E2 -1876.394} C_VEL
LIN {X 0,Y 580.971,Z 354.323,A -85,B 0,C 180,E1 -1876.445,E2 -1876.445} C_VEL
LIN {X 0,Y 580.813,Z 454.746,A -85,B 0,C 180,E1 -1877.709,E2 -1877.709} C_VEL
LIN {X 0,Y 580.752,Z 467.513,A -85,B 0,C 180,E1 -1877.995,E2 -1877.995} C_VEL
LIN {X 0,Y 580.635,Z 481.441,A -85,B 0,C 180,E1 -1878.48,E2 -1878.48} C_VEL
LIN {X 0,Y 580.567,Z 492.556,A -85,B 0,C 180,E1 -1879.009,E2 -1879.009} C_VEL
LIN {X 0,Y 580.452,Z 502.872,A -85,B 0,C 180,E1 -1879.624,E2 -1879.624} C_VEL
LIN {X 0,Y 580.358,Z 513.552,A -85,B 0,C 180,E1 -1880.415,E2 -1880.415} C_VEL
LIN {X 0,Y 580.271,Z 523.121,A -85,B 0,C 180,E1 -1881.292,E2 -1881.292} C_VEL
LIN {X 0,Y 580.221,Z 530.932,A -85,B 0,C 180,E1 -1882.168,E2 -1882.168} C_VEL
LIN {X 0,Y 580.157,Z 537.444,A -85,B 0,C 180,E1 -1883.042,E2 -1883.042} C_VEL
LIN {X 0,Y 580.162,Z 543.828,A -85,B 0,C 180,E1 -1884.09,E2 -1884.09} C_VEL
LIN {X 0,Y 580.053,Z 548.924,A -85,B 0,C 180,E1 -1885.135,E2 -1885.135} C_VEL
LIN {X 0,Y 580.109,Z 552.875,A -85,B 0,C 180,E1 -1886.18,E2 -1886.18} C_VEL
LIN {X 0,Y 580.043,Z 555.789,A -85,B 0,C 180,E1 -1887.222,E2 -1887.222} C_VEL
LIN {X 0,Y 580.047,Z 558.191,A -85,B 0,C 180,E1 -1888.611,E2 -1888.611} C_VEL
LIN {X 0,Y 580.04,Z 558.781,A -85,B 0,C 180,E1 -1889.306,E2 -1889.306} C_VEL
LIN {X 0,Y 580.04,Z 558.781,A -85,B 0,C 180,E1 -1890.694,E2 -1890.694} C_VEL
LIN {X 0,Y 580.047,Z 558.191,A -85,B 0,C 180,E1 -1891.389,E2 -1891.389} C_VEL
LIN {X 0,Y 580.043,Z 555.789,A -85,B 0,C 180,E1 -1892.778,E2 -1892.778} C_VEL
LIN {X 0,Y 580.109,Z 552.875,A -85,B 0,C 180,E1 -1893.82,E2 -1893.82} C_VEL
LIN {X 0,Y 580.053,Z 548.924,A -85,B 0,C 180,E1 -1894.865,E2 -1894.865} C_VEL
LIN {X 0,Y 580.162,Z 543.828,A -85,B 0,C 180,E1 -1895.91,E2 -1895.91} C_VEL
LIN {X 0,Y 580.157,Z 537.444,A -85,B 0,C 180,E1 -1896.958,E2 -1896.958} C_VEL
LIN {X 0,Y 580.242,Z 529.494,A -85,B 0,C 180,E1 -1898.007,E2 -1898.007} C_VEL
LIN {X 0,Y 580.304,Z 521.353,A -85,B 0,C 180,E1 -1898.883,E2 -1898.883} C_VEL
LIN {X 0,Y 580.353,Z 511.346,A -85,B 0,C 180,E1 -1899.761,E2 -1899.761} C_VEL
LIN {X 0,Y 580.483,Z 501.524,A -85,B 0,C 180,E1 -1900.463,E2 -1900.463} C_VEL
LIN {X 0,Y 580.578,Z 490.926,A -85,B 0,C 180,E1 -1901.079,E2 -1901.079} C_VEL
LIN {X 0,Y 580.657,Z 478.164,A -85,B 0,C 180,E1 -1901.652,E2 -1901.652} C_VEL
LIN {X 0,Y 580.742,Z 465.82,A -85,B 0,C 180,E1 -1902.049,E2 -1902.049} C_VEL
LIN {X 0,Y 580.813,Z 454.746,A -85,B 0,C 180,E1 -1902.291,E2 -1902.291} C_VEL
LIN {X 0,Y 580.849,Z 351.641,A -85,B 0,C 180,E1 -1903.591,E2 -1903.591} C_VEL
LIN {X 0,Y 580.389,Z 348.559,A -85,B 0,C 180,E1 -1903.658,E2 -1903.658} C_VEL
LIN {X 0,Y 580.326,Z 346.134,A -85,B 0,C 180,E1 -1904.017,E2 -1904.017} C_VEL
LIN {X 0,Y 580.452,Z 329.206,A -85,B 0,C 180,E1 -1906.958,E2 -1906.958} C_VEL
LIN {X 0,Y 580.641,Z 310.952,A -85,B 0,C 180,E1 -1910.179,E2 -1910.179} C_VEL
LIN {X 0,Y 580.785,Z 293.722,A -85,B 0,C 180,E1 -1913.275,E2 -1913.275} C_VEL
LIN {X 0,Y 580.741,Z 288.103,A -85,B 0,C 180,E1 -1914.296,E2 -1914.296} C_VEL
LIN {X 0,Y 580.294,Z 285.756,A -85,B 0,C 180,E1 -1914.786,E2 -1914.786} C_VEL
LIN {X 0,Y 580.288,Z 285.705,A -85,B 0,C 180,E1 -1917.856,E2 -1917.856} C_VEL
LIN {X 0,Y 580.281,Z 285.699,A -85,B 0,C 180,E1 -1920.693,E2 -1920.693} C_VEL
LIN {X 0,Y 580.302,Z 285.695,A -85,B 0,C 180,E1 -1923.315,E2 -1923.315} C_VEL
LIN {X 0,Y 580.242,Z 285.708,A -85,B 0,C 180,E1 -1925.755,E2 -1925.755} C_VEL
LIN {X 0,Y 580.282,Z 285.703,A -85,B 0,C 180,E1 -1928.146,E2 -1928.146} C_VEL
LIN {X 0,Y 580.293,Z 285.693,A -85,B 0,C 180,E1 -1930.843,E2 -1930.843} C_VEL
LIN {X 0,Y 580.275,Z 285.704,A -85,B 0,C 180,E1 -1933.657,E2 -1933.657} C_VEL
LIN {X 0,Y 580.272,Z 285.698,A -85,B 0,C 180,E1 -1936.608,E2 -1936.608} C_VEL
LIN {X 0,Y 580.296,Z 285.696,A -85,B 0,C 180,E1 -1939.156,E2 -1939.156} C_VEL
LIN {X 0,Y 580.284,Z 285.704,A -85,B 0,C 180,E1 -1941.926,E2 -1941.926} C_VEL
LIN {X 0,Y 580.249,Z 285.701,A -85,B 0,C 180,E1 -1944.452,E2 -1944.452} C_VEL
LIN {X 0,Y 580.283,Z 285.696,A -85,B 0,C 180,E1 -1946.974,E2 -1946.974} C_VEL
LIN {X 0,Y 580.288,Z 285.702,A -85,B 0,C 180,E1 -1949.424,E2 -1949.424} C_VEL
LIN {X 0,Y 580.313,Z 285.693,A -85,B 0,C 180,E1 -1952.136,E2 -1952.136} C_VEL
LIN {X 0,Y 580.312,Z 285.697,A -85,B 0,C 180,E1 -1955.269,E2 -1955.269} C_VEL
LIN {X 0,Y 580.263,Z 285.702,A -85,B 0,C 180,E1 -1957.947,E2 -1957.947} C_VEL
LIN {X 0,Y 580.309,Z 285.693,A -85,B 0,C 180,E1 -1960.913,E2 -1960.913} C_VEL
LIN {X 0,Y 580.271,Z 285.702,A -85,B 0,C 180,E1 -1963.825,E2 -1963.825} C_VEL
LIN {X 0,Y 580.316,Z 285.694,A -85,B 0,C 180,E1 -1965.982,E2 -1965.982} C_VEL
LIN {X 0,Y 580.322,Z 285.693,A -85,B 0,C 180,E1 -1968.827,E2 -1968.827} C_VEL
LIN {X 0,Y 580.324,Z 285.695,A -85,B 0,C 180,E1 -1971.643,E2 -1971.643} C_VEL
LIN {X 0,Y 580.317,Z 285.692,A -85,B 0,C 180,E1 -1974.44,E2 -1974.44} C_VEL
LIN {X 0,Y 580.336,Z 285.7,A -85,B 0,C 180,E1 -1977.223,E2 -1977.223} C_VEL
LIN {X 0,Y 580.335,Z 285.687,A -85,B 0,C 180,E1 -1980,E2 -1980} C_VEL
LIN {X 0,Y 580.34,Z 285.692,A -85,B 0,C 180,E1 -1982.776,E2 -1982.776} C_VEL
LIN {X 0,Y 580.316,Z 285.696,A -85,B 0,C 180,E1 -1985.559,E2 -1985.559} C_VEL
LIN {X 0,Y 580.323,Z 285.691,A -85,B 0,C 180,E1 -1988.356,E2 -1988.356} C_VEL
LIN {X 0,Y 580.322,Z 285.698,A -85,B 0,C 180,E1 -1991.208,E2 -1991.208} C_VEL
LIN {X 0,Y 580.304,Z 285.695,A -85,B 0,C 180,E1 -1994.339,E2 -1994.339} C_VEL
LIN {X 0,Y 580.303,Z 285.703,A -85,B 0,C 180,E1 -1996.915,E2 -1996.915} C_VEL
LIN {X 0,Y 580.297,Z 285.693,A -85,B 0,C 180,E1 -1999.822,E2 -1999.822} C_VEL
LIN {X 0,Y 580.276,Z 285.701,A -85,B 0,C 180,E1 -2001.345,E2 -2001.345} C_VEL
LIN {X 0,Y 579.578,Z 285.787,A -85,B 0,C 180,E1 -2001.925,E2 -2001.925} C_VEL
LIN {X 0,Y 576.701,Z 286.152,A -85,B 0,C 180,E1 -2002.864,E2 -2002.864} C_VEL
LIN {X 0,Y 574.306,Z 286.445,A -85,B 0,C 180,E1 -2003.621,E2 -2003.621} C_VEL
LIN {X 0,Y 573.308,Z 286.567,A -85,B 0,C 180,E1 -2004.204,E2 -2004.204} C_VEL
LIN {X 0,Y 573.241,Z 286.577,A -85,B 0,C 180,E1 -2004.402,E2 -2004.402} C_VEL
LIN {X 0,Y 573.241,Z 286.579,A -85,B 0,C 180,E1 -2006.976,E2 -2006.976} C_VEL
LIN {X 0,Y 573.243,Z 286.575,A -85,B 0,C 180,E1 -2009.49,E2 -2009.49} C_VEL
LIN {X 0,Y 573.246,Z 286.575,A -85,B 0,C 180,E1 -2012.229,E2 -2012.229} C_VEL
LIN {X 0,Y 573.244,Z 286.581,A -85,B 0,C 180,E1 -2014.774,E2 -2014.774} C_VEL
LIN {X 0,Y 573.245,Z 286.577,A -85,B 0,C 180,E1 -2017.167,E2 -2017.167} C_VEL
LIN {X 0,Y 573.241,Z 286.573,A -85,B 0,C 180,E1 -2019.607,E2 -2019.607} C_VEL
LIN {X 0,Y 573.234,Z 286.584,A -85,B 0,C 180,E1 -2022.642,E2 -2022.642} C_VEL
LIN {X 0,Y 573.23,Z 286.574,A -85,B 0,C 180,E1 -2025.667,E2 -2025.667} C_VEL
LIN {X 0,Y 573.238,Z 286.578,A -85,B 0,C 180,E1 -2028.545,E2 -2028.545} C_VEL
LIN {X 0,Y 573.241,Z 286.575,A -85,B 0,C 180,E1 -2031.299,E2 -2031.299} C_VEL
LIN {X 0,Y 573.257,Z 286.574,A -85,B 0,C 180,E1 -2034.012,E2 -2034.012} C_VEL
LIN {X 0,Y 573.278,Z 286.577,A -85,B 0,C 180,E1 -2036.519,E2 -2036.519} C_VEL
LIN {X 0,Y 573.232,Z 286.576,A -85,B 0,C 180,E1 -2039.116,E2 -2039.116} C_VEL
LIN {X 0,Y 573.259,Z 286.574,A -85,B 0,C 180,E1 -2041.969,E2 -2041.969} C_VEL
LIN {X 0,Y 573.253,Z 286.579,A -85,B 0,C 180,E1 -2044.591,E2 -2044.591} C_VEL
LIN {X 0,Y 573.232,Z 286.577,A -85,B 0,C 180,E1 -2047.663,E2 -2047.663} C_VEL
LIN {X 0,Y 573.274,Z 286.574,A -85,B 0,C 180,E1 -2050.729,E2 -2050.729} C_VEL
LIN {X 0,Y 573.248,Z 286.576,A -85,B 0,C 180,E1 -2053.622,E2 -2053.622} C_VEL
LIN {X 0,Y 573.269,Z 286.575,A -85,B 0,C 180,E1 -2055.807,E2 -2055.807} C_VEL
LIN {X 0,Y 573.259,Z 286.574,A -85,B 0,C 180,E1 -2058.745,E2 -2058.745} C_VEL
LIN {X 0,Y 573.282,Z 286.572,A -85,B 0,C 180,E1 -2061.541,E2 -2061.541} C_VEL
LIN {X 0,Y 573.291,Z 286.574,A -85,B 0,C 180,E1 -2064.372,E2 -2064.372} C_VEL
LIN {X 0,Y 573.313,Z 286.574,A -85,B 0,C 180,E1 -2067.892,E2 -2067.892} C_VEL
LIN {X 0,Y 573.329,Z 286.565,A -85,B 0,C 180,E1 -2070.702,E2 -2070.702} C_VEL
LIN {X 0,Y 573.302,Z 286.568,A -85,B 0,C 180,E1 -2072.811,E2 -2072.811} C_VEL
LIN {X 0,Y 573.291,Z 286.574,A -85,B 0,C 180,E1 -2075.628,E2 -2075.628} C_VEL
LIN {X 0,Y 573.282,Z 286.572,A -85,B 0,C 180,E1 -2078.459,E2 -2078.459} C_VEL
LIN {X 0,Y 573.268,Z 286.574,A -85,B 0,C 180,E1 -2081.312,E2 -2081.312} C_VEL
LIN {X 0,Y 573.278,Z 286.572,A -85,B 0,C 180,E1 -2084.424,E2 -2084.424} C_VEL
LIN {X 0,Y 573.255,Z 286.574,A -85,B 0,C 180,E1 -2087.111,E2 -2087.111} C_VEL
LIN {X 0,Y 573.249,Z 286.578,A -85,B 0,C 180,E1 -2090.076,E2 -2090.076} C_VEL
LIN {X 0,Y 573.229,Z 286.578,A -85,B 0,C 180,E1 -2093.099,E2 -2093.099} C_VEL
LIN {X 0,Y 573.253,Z 286.579,A -85,B 0,C 180,E1 -2095.409,E2 -2095.409} C_VEL
LIN {X 0,Y 573.259,Z 286.574,A -85,B 0,C 180,E1 -2098.031,E2 -2098.031} C_VEL
LIN {X 0,Y 573.232,Z 286.576,A -85,B 0,C 180,E1 -2100.884,E2 -2100.884} C_VEL
LIN {X 0,Y 573.282,Z 286.576,A -85,B 0,C 180,E1 -2103.528,E2 -2103.528} C_VEL
LIN {X 0,Y 573.254,Z 286.574,A -85,B 0,C 180,E1 -2106.048,E2 -2106.048} C_VEL
LIN {X 0,Y 573.241,Z 286.575,A -85,B 0,C 180,E1 -2108.701,E2 -2108.701} C_VEL
LIN {X 0,Y 573.246,Z 286.575,A -85,B 0,C 180,E1 -2111.595,E2 -2111.595} C_VEL
LIN {X 0,Y 573.23,Z 286.574,A -85,B 0,C 180,E1 -2114.333,E2 -2114.333} C_VEL
LIN {X 0,Y 573.234,Z 286.584,A -85,B 0,C 180,E1 -2117.358,E2 -2117.358} C_VEL
LIN {X 0,Y 573.241,Z 286.573,A -85,B 0,C 180,E1 -2120.393,E2 -2120.393} C_VEL
LIN {X 0,Y 573.247,Z 286.58,A -85,B 0,C 180,E1 -2123.078,E2 -2123.078} C_VEL
LIN {X 0,Y 573.266,Z 286.573,A -85,B 0,C 180,E1 -2125.672,E2 -2125.672} C_VEL
LIN {X 0,Y 573.24,Z 286.574,A -85,B 0,C 180,E1 -2128.185,E2 -2128.185} C_VEL
LIN {X 0,Y 573.26,Z 286.574,A -85,B 0,C 180,E1 -2130.634,E2 -2130.634} C_VEL
LIN {X 0,Y 573.241,Z 286.579,A -85,B 0,C 180,E1 -2133.024,E2 -2133.024} C_VEL
LIN {X 0,Y 573.265,Z 286.577,A -85,B 0,C 180,E1 -2135.366,E2 -2135.366} C_VEL
LIN {X 0,Y 573.221,Z 286.577,A -85,B 0,C 180,E1 -2138.419,E2 -2138.419} C_VEL
LIN {X 0,Y 573.269,Z 286.573,A -85,B 0,C 180,E1 -2140.728,E2 -2140.728} C_VEL
LIN {X 0,Y 573.249,Z 286.574,A -85,B 0,C 180,E1 -2143.622,E2 -2143.622} C_VEL
LIN {X 0,Y 573.228,Z 286.579,A -85,B 0,C 180,E1 -2146.53,E2 -2146.53} C_VEL
LIN {X 0,Y 573.272,Z 286.575,A -85,B 0,C 180,E1 -2148.734,E2 -2148.734} C_VEL
LIN {X 0,Y 573.28,Z 286.569,A -85,B 0,C 180,E1 -2151.541,E2 -2151.541} C_VEL
LIN {X 0,Y 573.282,Z 286.572,A -85,B 0,C 180,E1 -2154.372,E2 -2154.372} C_VEL
LIN {X 0,Y 573.305,Z 286.568,A -85,B 0,C 180,E1 -2157.19,E2 -2157.19} C_VEL
LIN {X 0,Y 573.305,Z 286.561,A -85,B 0,C 180,E1 -2160,E2 -2160} C_VEL
LIN {X 0,Y 573.302,Z 286.575,A -85,B 0,C 180,E1 -2162.811,E2 -2162.811} C_VEL
LIN {X 0,Y 573.283,Z 286.568,A -85,B 0,C 180,E1 -2165.629,E2 -2165.629} C_VEL
LIN {X 0,Y 573.297,Z 286.572,A -85,B 0,C 180,E1 -2168.46,E2 -2168.46} C_VEL
LIN {X 0,Y 573.29,Z 286.567,A -85,B 0,C 180,E1 -2171.312,E2 -2171.312} C_VEL
LIN {X 0,Y 573.271,Z 286.577,A -85,B 0,C 180,E1 -2174.425,E2 -2174.425} C_VEL
LIN {X 0,Y 573.249,Z 286.572,A -85,B 0,C 180,E1 -2177.112,E2 -2177.112} C_VEL
LIN {X 0,Y 573.248,Z 286.574,A -85,B 0,C 180,E1 -2180.077,E2 -2180.077} C_VEL
LIN {X 0,Y 573.228,Z 286.583,A -85,B 0,C 180,E1 -2182.339,E2 -2182.339} C_VEL
LIN {X 0,Y 573.244,Z 286.572,A -85,B 0,C 180,E1 -2185.411,E2 -2185.411} C_VEL
LIN {X 0,Y 573.258,Z 286.574,A -85,B 0,C 180,E1 -2188.033,E2 -2188.033} C_VEL
LIN {X 0,Y 573.221,Z 286.579,A -85,B 0,C 180,E1 -2190.883,E2 -2190.883} C_VEL
LIN {X 0,Y 573.234,Z 286.573,A -85,B 0,C 180,E1 -2193.522,E2 -2193.522} C_VEL
LIN {X 0,Y 573.209,Z 286.583,A -85,B 0,C 180,E1 -2196.052,E2 -2196.052} C_VEL
LIN {X 0,Y 573.236,Z 286.577,A -85,B 0,C 180,E1 -2198.702,E2 -2198.702} C_VEL
LIN {X 0,Y 573.238,Z 286.576,A -85,B 0,C 180,E1 -2201.595,E2 -2201.595} C_VEL
LIN {X 0,Y 573.228,Z 286.583,A -85,B 0,C 180,E1 -2204.335,E2 -2204.335} C_VEL
LIN {X 0,Y 573.233,Z 286.576,A -85,B 0,C 180,E1 -2207.36,E2 -2207.36} C_VEL
LIN {X 0,Y 573.235,Z 286.58,A -85,B 0,C 180,E1 -2210.393,E2 -2210.393} C_VEL
LIN {X 0,Y 573.229,Z 286.575,A -85,B 0,C 180,E1 -2213.077,E2 -2213.077} C_VEL
LIN {X 0,Y 573.263,Z 286.576,A -85,B 0,C 180,E1 -2215.672,E2 -2215.672} C_VEL
LIN {X 0,Y 573.236,Z 286.582,A -85,B 0,C 180,E1 -2218.185,E2 -2218.185} C_VEL
LIN {X 0,Y 573.26,Z 286.574,A -85,B 0,C 180,E1 -2220.635,E2 -2220.635} C_VEL
LIN {X 0,Y 573.213,Z 286.58,A -85,B 0,C 180,E1 -2223.023,E2 -2223.023} C_VEL
LIN {X 0,Y 573.267,Z 286.75,A -85,B 0,C 180,E1 -2225.123,E2 -2225.123} C_VEL
LIN {X 0,Y 573.844,Z 291.114,A -85,B 0,C 180,E1 -2225.97,E2 -2225.97} C_VEL
LIN {X 0,Y 573.684,Z 307.236,A -85,B 0,C 180,E1 -2228.892,E2 -2228.892} C_VEL
LIN {X 0,Y 573.488,Z 323.369,A -85,B 0,C 180,E1 -2231.791,E2 -2231.791} C_VEL
LIN {X 0,Y 573.364,Z 338.891,A -85,B 0,C 180,E1 -2234.538,E2 -2234.538} C_VEL
LIN {X 0,Y 573.309,Z 348.251,A -85,B 0,C 180,E1 -2236.148,E2 -2236.148} C_VEL
LIN {X 0,Y 573.627,Z 350.341,A -85,B 0,C 180,E1 -2236.218,E2 -2236.218} C_VEL
LIN {X 0,Y 574.076,Z 354.323,A -85,B 0,C 180,E1 -2236.279,E2 -2236.279} C_VEL
LIN {X 0,Y 573.892,Z 454.69,A -85,B 0,C 180,E1 -2237.558,E2 -2237.558} C_VEL
LIN {X 0,Y 573.805,Z 467.513,A -85,B 0,C 180,E1 -2237.848,E2 -2237.848} C_VEL
LIN {X 0,Y 573.684,Z 481.422,A -85,B 0,C 180,E1 -2238.339,E2 -2238.339} C_VEL
LIN {X 0,Y 573.576,Z 492.64,A -85,B 0,C 180,E1 -2238.879,E2 -2238.879} C_VEL
LIN {X 0,Y 573.471,Z 502.856,A -85,B 0,C 180,E1 -2239.497,E2 -2239.497} C_VEL
LIN {X 0,Y 573.336,Z 513.556,A -85,B 0,C 180,E1 -2240.297,E2 -2240.297} C_VEL
LIN {X 0,Y 573.24,Z 523.118,A -85,B 0,C 180,E1 -2241.185,E2 -2241.185} C_VEL
LIN {X 0,Y 573.161,Z 530.923,A -85,B 0,C 180,E1 -2242.071,E2 -2242.071} C_VEL
LIN {X 0,Y 573.082,Z 537.435,A -85,B 0,C 180,E1 -2242.956,E2 -2242.956} C_VEL
LIN {X 0,Y 573.074,Z 543.819,A -85,B 0,C 180,E1 -2244.017,E2 -2244.017} C_VEL
LIN {X 0,Y 572.962,Z 548.915,A -85,B 0,C 180,E1 -2245.074,E2 -2245.074} C_VEL
LIN {X 0,Y 573.014,Z 552.867,A -85,B 0,C 180,E1 -2246.132,E2 -2246.132} C_VEL
LIN {X 0,Y 572.959,Z 555.784,A -85,B 0,C 180,E1 -2247.188,E2 -2247.188} C_VEL
LIN {X 0,Y 572.946,Z 558.192,A -85,B 0,C 180,E1 -2248.594,E2 -2248.594} C_VEL
LIN {X 0,Y 572.941,Z 558.781,A -85,B 0,C 180,E1 -2249.297,E2 -2249.297} C_VEL
LIN {X 0,Y 572.941,Z 558.781,A -85,B 0,C 180,E1 -2250.703,E2 -2250.703} C_VEL
LIN {X 0,Y 572.946,Z 558.192,A -85,B 0,C 180,E1 -2251.406,E2 -2251.406} C_VEL
LIN {X 0,Y 572.959,Z 555.784,A -85,B 0,C 180,E1 -2252.812,E2 -2252.812} C_VEL
LIN {X 0,Y 573.014,Z 552.867,A -85,B 0,C 180,E1 -2253.868,E2 -2253.868} C_VEL
LIN {X 0,Y 572.962,Z 548.915,A -85,B 0,C 180,E1 -2254.926,E2 -2254.926} C_VEL
LIN {X 0,Y 573.074,Z 543.819,A -85,B 0,C 180,E1 -2255.983,E2 -2255.983} C_VEL
LIN {X 0,Y 573.082,Z 537.435,A -85,B 0,C 180,E1 -2257.044,E2 -2257.044} C_VEL
LIN {X 0,Y 573.177,Z 529.498,A -85,B 0,C 180,E1 -2258.106,E2 -2258.106} C_VEL
LIN {X 0,Y 573.279,Z 521.357,A -85,B 0,C 180,E1 -2258.992,E2 -2258.992} C_VEL
LIN {X 0,Y 573.337,Z 511.332,A -85,B 0,C 180,E1 -2259.881,E2 -2259.881} C_VEL
LIN {X 0,Y 573.495,Z 501.507,A -85,B 0,C 180,E1 -2260.592,E2 -2260.592} C_VEL
LIN {X 0,Y 573.623,Z 490.293,A -85,B 0,C 180,E1 -2261.249,E2 -2261.249} C_VEL
LIN {X 0,Y 573.705,Z 476.945,A -85,B 0,C 180,E1 -2261.84,E2 -2261.84} C_VEL
LIN {X 0,Y 573.836,Z 464.912,A -85,B 0,C 180,E1 -2262.219,E2 -2262.219} C_VEL
LIN {X 0,Y 573.898,Z 453.359,A -85,B 0,C 180,E1 -2262.464,E2 -2262.464} C_VEL
LIN {X 0,Y 573.946,Z 352.334,A -85,B 0,C 180,E1 -2263.749,E2 -2263.749} C_VEL
LIN {X 0,Y 573.347,Z 348.571,A -85,B 0,C 180,E1 -2263.829,E2 -2263.829} C_VEL
LIN {X 0,Y 573.287,Z 346.134,A -85,B 0,C 180,E1 -2264.192,E2 -2264.192} C_VEL
LIN {X 0,Y 573.432,Z 331.743,A -85,B 0,C 180,E1 -2266.722,E2 -2266.722} C_VEL
LIN {X 0,Y 573.579,Z 316.951,A -85,B 0,C 180,E1 -2269.356,E2 -2269.356} C_VEL
LIN {X 0,Y 573.712,Z 301.569,A -85,B 0,C 180,E1 -2272.128,E2 -2272.128} C_VEL
LIN {X 0,Y 573.826,Z 290.093,A -85,B 0,C 180,E1 -2274.223,E2 -2274.223} C_VEL
LIN {X 0,Y 573.249,Z 286.615,A -85,B 0,C 180,E1 -2274.95,E2 -2274.95} C_VEL
LIN {X 0,Y 573.263,Z 286.579,A -85,B 0,C 180,E1 -2277.766,E2 -2277.766} C_VEL
LIN {X 0,Y 573.243,Z 286.583,A -85,B 0,C 180,E1 -2280.175,E2 -2280.175} C_VEL
LIN {X 0,Y 573.25,Z 286.574,A -85,B 0,C 180,E1 -2282.644,E2 -2282.644} C_VEL
LIN {X 0,Y 573.203,Z 286.579,A -85,B 0,C 180,E1 -2285.187,E2 -2285.187} C_VEL
LIN {X 0,Y 573.228,Z 286.583,A -85,B 0,C 180,E1 -2287.807,E2 -2287.807} C_VEL
LIN {X 0,Y 573.241,Z 286.572,A -85,B 0,C 180,E1 -2290.524,E2 -2290.524} C_VEL
LIN {X 0,Y 573.235,Z 286.577,A -85,B 0,C 180,E1 -2293.358,E2 -2293.358} C_VEL
LIN {X 0,Y 573.239,Z 286.577,A -85,B 0,C 180,E1 -2296.33,E2 -2296.33} C_VEL
LIN {X 0,Y 573.269,Z 286.575,A -85,B 0,C 180,E1 -2299.477,E2 -2299.477} C_VEL
LIN {X 0,Y 573.23,Z 286.579,A -85,B 0,C 180,E1 -2302.192,E2 -2302.192} C_VEL
LIN {X 0,Y 573.233,Z 286.577,A -85,B 0,C 180,E1 -2305.227,E2 -2305.227} C_VEL
LIN {X 0,Y 573.234,Z 286.577,A -85,B 0,C 180,E1 -2308.184,E2 -2308.184} C_VEL
LIN {X 0,Y 573.256,Z 286.572,A -85,B 0,C 180,E1 -2310.633,E2 -2310.633} C_VEL
LIN {X 0,Y 573.244,Z 286.573,A -85,B 0,C 180,E1 -2313.023,E2 -2313.023} C_VEL
LIN {X 0,Y 573.266,Z 286.576,A -85,B 0,C 180,E1 -2315.365,E2 -2315.365} C_VEL
LIN {X 0,Y 573.222,Z 286.576,A -85,B 0,C 180,E1 -2318.419,E2 -2318.419} C_VEL
LIN {X 0,Y 573.271,Z 286.568,A -85,B 0,C 180,E1 -2320.727,E2 -2320.727} C_VEL
LIN {X 0,Y 573.248,Z 286.579,A -85,B 0,C 180,E1 -2323.621,E2 -2323.621} C_VEL
LIN {X 0,Y 573.23,Z 286.575,A -85,B 0,C 180,E1 -2326.529,E2 -2326.529} C_VEL
LIN {X 0,Y 573.274,Z 286.569,A -85,B 0,C 180,E1 -2328.734,E2 -2328.734} C_VEL
LIN {X 0,Y 573.297,Z 286.572,A -85,B 0,C 180,E1 -2331.54,E2 -2331.54} C_VEL
LIN {X 0,Y 573.283,Z 286.568,A -85,B 0,C 180,E1 -2334.371,E2 -2334.371} C_VEL
LIN {X 0,Y 573.302,Z 286.575,A -85,B 0,C 180,E1 -2337.189,E2 -2337.189} C_VEL
LIN {X 0,Y 573.305,Z 286.561,A -85,B 0,C 180,E1 -2340,E2 -2340} C_VEL
LIN {X 0,Y 573.305,Z 286.568,A -85,B 0,C 180,E1 -2342.81,E2 -2342.81} C_VEL
LIN {X 0,Y 573.282,Z 286.572,A -85,B 0,C 180,E1 -2345.628,E2 -2345.628} C_VEL
LIN {X 0,Y 573.28,Z 286.569,A -85,B 0,C 180,E1 -2348.459,E2 -2348.459} C_VEL
LIN {X 0,Y 573.288,Z 286.573,A -85,B 0,C 180,E1 -2351.311,E2 -2351.311} C_VEL
LIN {X 0,Y 573.27,Z 286.572,A -85,B 0,C 180,E1 -2354.424,E2 -2354.424} C_VEL
LIN {X 0,Y 573.248,Z 286.579,A -85,B 0,C 180,E1 -2357.111,E2 -2357.111} C_VEL
LIN {X 0,Y 573.246,Z 286.571,A -85,B 0,C 180,E1 -2360.076,E2 -2360.076} C_VEL
LIN {X 0,Y 573.227,Z 286.577,A -85,B 0,C 180,E1 -2362.338,E2 -2362.338} C_VEL
LIN {X 0,Y 573.241,Z 286.577,A -85,B 0,C 180,E1 -2364.402,E2 -2364.402} C_VEL
LIN {X 0,Y 572.614,Z 286.661,A -85,B 0,C 180,E1 -2364.988,E2 -2364.988} C_VEL
LIN {X 0,Y 569.771,Z 287.015,A -85,B 0,C 180,E1 -2365.94,E2 -2365.94} C_VEL
LIN {X 0,Y 567.34,Z 287.315,A -85,B 0,C 180,E1 -2366.705,E2 -2366.705} C_VEL
LIN {X 0,Y 566.289,Z 287.44,A -85,B 0,C 180,E1 -2367.297,E2 -2367.297} C_VEL
LIN {X 0,Y 566.201,Z 287.449,A -85,B 0,C 180,E1 -2367.497,E2 -2367.497} C_VEL
LIN {X 0,Y 566.217,Z 287.449,A -85,B 0,C 180,E1 -2369.767,E2 -2369.767} C_VEL
LIN {X 0,Y 566.198,Z 287.456,A -85,B 0,C 180,E1 -2372.431,E2 -2372.431} C_VEL
LIN {X 0,Y 566.205,Z 287.455,A -85,B 0,C 180,E1 -2374.995,E2 -2374.995} C_VEL
LIN {X 0,Y 566.187,Z 287.454,A -85,B 0,C 180,E1 -2377.461,E2 -2377.461} C_VEL
LIN {X 0,Y 566.218,Z 287.451,A -85,B 0,C 180,E1 -2380.198,E2 -2380.198} C_VEL
LIN {X 0,Y 566.196,Z 287.455,A -85,B 0,C 180,E1 -2383.054,E2 -2383.054} C_VEL
LIN {X 0,Y 566.193,Z 287.452,A -85,B 0,C 180,E1 -2386.049,E2 -2386.049} C_VEL
LIN {X 0,Y 566.204,Z 287.453,A -85,B 0,C 180,E1 -2388.864,E2 -2388.864} C_VEL
LIN {X 0,Y 566.182,Z 287.454,A -85,B 0,C 180,E1 -2391.638,E2 -2391.638} C_VEL
LIN {X 0,Y 566.205,Z 287.457,A -85,B 0,C 180,E1 -2394.312,E2 -2394.312} C_VEL
LIN {X 0,Y 566.223,Z 287.451,A -85,B 0,C 180,E1 -2396.899,E2 -2396.899} C_VEL
LIN {X 0,Y 566.182,Z 287.453,A -85,B 0,C 180,E1 -2399.408,E2 -2399.408} C_VEL
LIN {X 0,Y 566.223,Z 287.449,A -85,B 0,C 180,E1 -2401.859,E2 -2401.859} C_VEL
LIN {X 0,Y 566.221,Z 287.458,A -85,B 0,C 180,E1 -2404.252,E2 -2404.252} C_VEL
LIN {X 0,Y 566.186,Z 287.457,A -85,B 0,C 180,E1 -2406.714,E2 -2406.714} C_VEL
LIN {X 0,Y 566.21,Z 287.452,A -85,B 0,C 180,E1 -2409.663,E2 -2409.663} C_VEL
LIN {X 0,Y 566.199,Z 287.456,A -85,B 0,C 180,E1 -2412.669,E2 -2412.669} C_VEL
LIN {X 0,Y 566.23,Z 287.45,A -85,B 0,C 180,E1 -2415.627,E2 -2415.627} C_VEL
LIN {X 0,Y 566.231,Z 287.451,A -85,B 0,C 180,E1 -2418.675,E2 -2418.675} C_VEL
LIN {X 0,Y 566.226,Z 287.45,A -85,B 0,C 180,E1 -2421.434,E2 -2421.434} C_VEL
LIN {X 0,Y 566.259,Z 287.451,A -85,B 0,C 180,E1 -2424.302,E2 -2424.302} C_VEL
LIN {X 0,Y 566.283,Z 287.449,A -85,B 0,C 180,E1 -2427.866,E2 -2427.866} C_VEL
LIN {X 0,Y 566.3,Z 287.441,A -85,B 0,C 180,E1 -2430.711,E2 -2430.711} C_VEL
LIN {X 0,Y 566.269,Z 287.444,A -85,B 0,C 180,E1 -2432.846,E2 -2432.846} C_VEL
LIN {X 0,Y 566.259,Z 287.451,A -85,B 0,C 180,E1 -2435.698,E2 -2435.698} C_VEL
LIN {X 0,Y 566.226,Z 287.45,A -85,B 0,C 180,E1 -2438.566,E2 -2438.566} C_VEL
LIN {X 0,Y 566.238,Z 287.451,A -85,B 0,C 180,E1 -2441.454,E2 -2441.454} C_VEL
LIN {X 0,Y 566.23,Z 287.449,A -85,B 0,C 180,E1 -2444.507,E2 -2444.507} C_VEL
LIN {X 0,Y 566.199,Z 287.455,A -85,B 0,C 180,E1 -2447.331,E2 -2447.331} C_VEL
LIN {X 0,Y 566.21,Z 287.452,A -85,B 0,C 180,E1 -2450.337,E2 -2450.337} C_VEL
LIN {X 0,Y 566.184,Z 287.459,A -85,B 0,C 180,E1 -2453.403,E2 -2453.403} C_VEL
LIN {X 0,Y 566.221,Z 287.458,A -85,B 0,C 180,E1 -2455.748,E2 -2455.748} C_VEL
LIN {X 0,Y 566.201,Z 287.452,A -85,B 0,C 180,E1 -2458.203,E2 -2458.203} C_VEL
LIN {X 0,Y 566.193,Z 287.454,A -85,B 0,C 180,E1 -2461.078,E2 -2461.078} C_VEL
LIN {X 0,Y 566.222,Z 287.45,A -85,B 0,C 180,E1 -2463.736,E2 -2463.736} C_VEL
LIN {X 0,Y 566.209,Z 287.449,A -85,B 0,C 180,E1 -2466.568,E2 -2466.568} C_VEL
LIN {X 0,Y 566.205,Z 287.454,A -85,B 0,C 180,E1 -2469.685,E2 -2469.685} C_VEL
LIN {X 0,Y 566.206,Z 287.445,A -85,B 0,C 180,E1 -2472.087,E2 -2472.087} C_VEL
LIN {X 0,Y 566.165,Z 287.458,A -85,B 0,C 180,E1 -2475.035,E2 -2475.035} C_VEL
LIN {X 0,Y 566.209,Z 287.449,A -85,B 0,C 180,E1 -2478.135,E2 -2478.135} C_VEL
LIN {X 0,Y 566.214,Z 287.45,A -85,B 0,C 180,E1 -2480.727,E2 -2480.727} C_VEL
LIN {X 0,Y 566.209,Z 287.451,A -85,B 0,C 180,E1 -2483.783,E2 -2483.783} C_VEL
LIN {X 0,Y 566.219,Z 287.447,A -85,B 0,C 180,E1 -2486.263,E2 -2486.263} C_VEL
LIN {X 0,Y 566.193,Z 287.457,A -85,B 0,C 180,E1 -2488.921,E2 -2488.921} C_VEL
LIN {X 0,Y 566.187,Z 287.46,A -85,B 0,C 180,E1 -2491.047,E2 -2491.047} C_VEL
LIN {X 0,Y 566.206,Z 287.454,A -85,B 0,C 180,E1 -2493.459,E2 -2493.459} C_VEL
LIN {X 0,Y 566.189,Z 287.453,A -85,B 0,C 180,E1 -2495.819,E2 -2495.819} C_VEL
LIN {X 0,Y 566.206,Z 287.457,A -85,B 0,C 180,E1 -2498.903,E2 -2498.903} C_VEL
LIN {X 0,Y 566.202,Z 287.456,A -85,B 0,C 180,E1 -2501.173,E2 -2501.173} C_VEL
LIN {X 0,Y 566.211,Z 287.453,A -85,B 0,C 180,E1 -2503.413,E2 -2503.413} C_VEL
LIN {X 0,Y 566.19,Z 287.454,A -85,B 0,C 180,E1 -2506.359,E2 -2506.359} C_VEL
LIN {X 0,Y 566.264,Z 287.447,A -85,B 0,C 180,E1 -2508.654,E2 -2508.654} C_VEL
LIN {X 0,Y 566.224,Z 287.448,A -85,B 0,C 180,E1 -2511.435,E2 -2511.435} C_VEL
LIN {X 0,Y 566.249,Z 287.447,A -85,B 0,C 180,E1 -2514.302,E2 -2514.302} C_VEL
LIN {X 0,Y 566.266,Z 287.441,A -85,B 0,C 180,E1 -2517.867,E2 -2517.867} C_VEL
LIN {X 0,Y 566.3,Z 287.442,A -85,B 0,C 180,E1 -2520.711,E2 -2520.711} C_VEL
LIN {X 0,Y 566.184,Z 287.453,A -85,B 0,C 180,E1 -2523.559,E2 -2523.559} C_VEL
LIN {X 0,Y 566.25,Z 287.444,A -85,B 0,C 180,E1 -2525.699,E2 -2525.699} C_VEL
LIN {X 0,Y 566.238,Z 287.452,A -85,B 0,C 180,E1 -2528.566,E2 -2528.566} C_VEL
LIN {X 0,Y 566.242,Z 287.444,A -85,B 0,C 180,E1 -2531.455,E2 -2531.455} C_VEL
LIN {X 0,Y 566.224,Z 287.457,A -85,B 0,C 180,E1 -2534.507,E2 -2534.507} C_VEL
LIN {X 0,Y 566.191,Z 287.449,A -85,B 0,C 180,E1 -2537.332,E2 -2537.332} C_VEL
LIN {X 0,Y 566.211,Z 287.454,A -85,B 0,C 180,E1 -2540.338,E2 -2540.338} C_VEL
LIN {X 0,Y 566.164,Z 287.456,A -85,B 0,C 180,E1 -2543.283,E2 -2543.283} C_VEL
LIN {X 0,Y 566.204,Z 287.45,A -85,B 0,C 180,E1 -2545.75,E2 -2545.75} C_VEL
LIN {X 0,Y 566.2,Z 287.455,A -85,B 0,C 180,E1 -2548.204,E2 -2548.204} C_VEL
LIN {X 0,Y 566.184,Z 287.454,A -85,B 0,C 180,E1 -2551.077,E2 -2551.077} C_VEL
LIN {X 0,Y 566.191,Z 287.452,A -85,B 0,C 180,E1 -2553.733,E2 -2553.733} C_VEL
LIN {X 0,Y 566.194,Z 287.457,A -85,B 0,C 180,E1 -2556.571,E2 -2556.571} C_VEL
LIN {X 0,Y 566.209,Z 287.451,A -85,B 0,C 180,E1 -2559.687,E2 -2559.687} C_VEL
LIN {X 0,Y 566.206,Z 287.458,A -85,B 0,C 180,E1 -2562.088,E2 -2562.088} C_VEL
LIN {X 0,Y 566.165,Z 287.455,A -85,B 0,C 180,E1 -2565.037,E2 -2565.037} C_VEL
LIN {X 0,Y 566.184,Z 287.46,A -85,B 0,C 180,E1 -2567.911,E2 -2567.911} C_VEL
LIN {X 0,Y 566.21,Z 287.451,A -85,B 0,C 180,E1 -2570.727,E2 -2570.727} C_VEL
LIN {X 0,Y 566.179,Z 287.455,A -85,B 0,C 180,E1 -2573.43,E2 -2573.43} C_VEL
LIN {X 0,Y 566.21,Z 287.455,A -85,B 0,C 180,E1 -2576.267,E2 -2576.267} C_VEL
LIN {X 0,Y 566.188,Z 287.454,A -85,B 0,C 180,E1 -2578.925,E2 -2578.925} C_VEL
LIN {X 0,Y 566.191,Z 287.461,A -85,B 0,C 180,E1 -2581.857,E2 -2581.857} C_VEL
LIN {X 0,Y 566.237,Z 287.502,A -85,B 0,C 180,E1 -2584.93,E2 -2584.93} C_VEL
LIN {X 0,Y 566.903,Z 292.063,A -85,B 0,C 180,E1 -2585.852,E2 -2585.852} C_VEL
LIN {X 0,Y 566.707,Z 307.467,A -85,B 0,C 180,E1 -2588.686,E2 -2588.686} C_VEL
LIN {X 0,Y 566.486,Z 322.334,A -85,B 0,C 180,E1 -2591.37,E2 -2591.37} C_VEL
LIN {X 0,Y 566.389,Z 335.786,A -85,B 0,C 180,E1 -2593.789,E2 -2593.789} C_VEL
LIN {X 0,Y 566.28,Z 348.258,A -85,B 0,C 180,E1 -2595.972,E2 -2595.972} C_VEL
LIN {X 0,Y 566.609,Z 350.451,A -85,B 0,C 180,E1 -2596.045,E2 -2596.045} C_VEL
LIN {X 0,Y 567.206,Z 354.323,A -85,B 0,C 180,E1 -2596.11,E2 -2596.11} C_VEL
LIN {X 0,Y 566.957,Z 454.634,A -85,B 0,C 180,E1 -2597.403,E2 -2597.403} C_VEL
LIN {X 0,Y 566.881,Z 466.626,A -85,B 0,C 180,E1 -2597.674,E2 -2597.674} C_VEL
LIN {X 0,Y 566.745,Z 480.393,A -85,B 0,C 180,E1 -2598.149,E2 -2598.149} C_VEL
LIN {X 0,Y 566.606,Z 492.041,A -85,B 0,C 180,E1 -2598.708,E2 -2598.708} C_VEL
LIN {X 0,Y 566.514,Z 501.491,A -85,B 0,C 180,E1 -2599.276,E2 -2599.276} C_VEL
LIN {X 0,Y 566.374,Z 510.188,A -85,B 0,C 180,E1 -2599.906,E2 -2599.906} C_VEL
LIN {X 0,Y 566.301,Z 517.553,A -85,B 0,C 180,E1 -2600.536,E2 -2600.536} C_VEL
LIN {X 0,Y 566.159,Z 524.739,A -85,B 0,C 180,E1 -2601.254,E2 -2601.254} C_VEL
LIN {X 0,Y 566.094,Z 532.285,A -85,B 0,C 180,E1 -2602.151,E2 -2602.151} C_VEL
LIN {X 0,Y 566.004,Z 538.691,A -85,B 0,C 180,E1 -2603.065,E2 -2603.065} C_VEL
LIN {X 0,Y 565.989,Z 543.809,A -85,B 0,C 180,E1 -2603.942,E2 -2603.942} C_VEL
LIN {X 0,Y 565.877,Z 548.906,A -85,B 0,C 180,E1 -2605.013,E2 -2605.013} C_VEL
LIN {X 0,Y 565.926,Z 552.86,A -85,B 0,C 180,E1 -2606.084,E2 -2606.084} C_VEL
LIN {X 0,Y 565.878,Z 555.779,A -85,B 0,C 180,E1 -2607.153,E2 -2607.153} C_VEL
LIN {X 0,Y 565.846,Z 558.194,A -85,B 0,C 180,E1 -2608.577,E2 -2608.577} C_VEL
LIN {X 0,Y 565.841,Z 558.781,A -85,B 0,C 180,E1 -2609.288,E2 -2609.288} C_VEL
LIN {X 0,Y 565.841,Z 558.781,A -85,B 0,C 180,E1 -2610.712,E2 -2610.712} C_VEL
LIN {X 0,Y 565.846,Z 558.194,A -85,B 0,C 180,E1 -2611.423,E2 -2611.423} C_VEL
LIN {X 0,Y 565.878,Z 555.779,A -85,B 0,C 180,E1 -2612.847,E2 -2612.847} C_VEL
LIN {X 0,Y 565.926,Z 552.86,A -85,B 0,C 180,E1 -2613.916,E2 -2613.916} C_VEL
LIN {X 0,Y 565.877,Z 548.906,A -85,B 0,C 180,E1 -2614.987,E2 -2614.987} C_VEL
LIN {X 0,Y 565.99,Z 543.809,A -85,B 0,C 180,E1 -2616.058,E2 -2616.058} C_VEL
LIN {X 0,Y 566.032,Z 537.426,A -85,B 0,C 180,E1 -2617.132,E2 -2617.132} C_VEL
LIN {X 0,Y 566.131,Z 529.501,A -85,B 0,C 180,E1 -2618.207,E2 -2618.207} C_VEL
LIN {X 0,Y 566.237,Z 521.36,A -85,B 0,C 180,E1 -2619.105,E2 -2619.105} C_VEL
LIN {X 0,Y 566.324,Z 511.319,A -85,B 0,C 180,E1 -2620.005,E2 -2620.005} C_VEL
LIN {X 0,Y 566.487,Z 502.84,A -85,B 0,C 180,E1 -2620.634,E2 -2620.634} C_VEL
LIN {X 0,Y 566.611,Z 493.284,A -85,B 0,C 180,E1 -2621.223,E2 -2621.223} C_VEL
LIN {X 0,Y 566.725,Z 483.612,A -85,B 0,C 180,E1 -2621.707,E2 -2621.707} C_VEL
LIN {X 0,Y 566.794,Z 474.35,A -85,B 0,C 180,E1 -2622.078,E2 -2622.078} C_VEL
LIN {X 0,Y 566.903,Z 463.131,A -85,B 0,C 180,E1 -2622.416,E2 -2622.416} C_VEL
LIN {X 0,Y 566.995,Z 450.621,A -85,B 0,C 180,E1 -2622.664,E2 -2622.664} C_VEL
LIN {X 0,Y 567.079,Z 353.229,A -85,B 0,C 180,E1 -2623.907,E2 -2623.907} C_VEL
LIN {X 0,Y 566.319,Z 348.583,A -85,B 0,C 180,E1 -2624.004,E2 -2624.004} C_VEL
LIN {X 0,Y 566.267,Z 347.169,A -85,B 0,C 180,E1 -2624.189,E2 -2624.189} C_VEL
LIN {X 0,Y 566.443,Z 330.356,A -85,B 0,C 180,E1 -2627.184,E2 -2627.184} C_VEL
LIN {X 0,Y 566.673,Z 312.951,A -85,B 0,C 180,E1 -2630.319,E2 -2630.319} C_VEL
LIN {X 0,Y 566.851,Z 296.244,A -85,B 0,C 180,E1 -2633.374,E2 -2633.374} C_VEL
LIN {X 0,Y 566.844,Z 291.041,A -85,B 0,C 180,E1 -2634.346,E2 -2634.346} C_VEL
LIN {X 0,Y 566.227,Z 287.486,A -85,B 0,C 180,E1 -2635.093,E2 -2635.093} C_VEL
LIN {X 0,Y 566.203,Z 287.459,A -85,B 0,C 180,E1 -2638.201,E2 -2638.201} C_VEL
